LIN {X 0,Y 186.284,Z 510.696,A -85,B 0,C 180,E1 -23810.819,E2 -23810.819} C_VEL
LIN {X 0,Y 183.87,Z 513.938,A -85,B 0,C 180,E1 -23812.309,E2 -23812.309} C_VEL
LIN {X 0,Y 178.035,Z 519.948,A -85,B 0,C 180,E1 -23815.094,E2 -23815.094} C_VEL
LIN {X 0,Y 171.013,Z 526.327,A -85,B 0,C 180,E1 -23819.1,E2 -23819.1} C_VEL
LIN {X 0,Y 166.228,Z 530.269,A -85,B 0,C 180,E1 -23822.61,E2 -23822.61} C_VEL
LIN {X 0,Y 161.84,Z 533.649,A -85,B 0,C 180,E1 -23827.005,E2 -23827.005} C_VEL
LIN {X 0,Y 158.22,Z 535.815,A -85,B 0,C 180,E1 -23831.895,E2 -23831.895} C_VEL
LIN {X 0,Y 156.037,Z 536.613,A -85,B 0,C 180,E1 -23836.995,E2 -23836.995} C_VEL
LIN {X 0,Y 155.154,Z 536.037,A -85,B 0,C 180,E1 -23842.2,E2 -23842.2} C_VEL
LIN {X 0,Y 155.187,Z 535.075,A -85,B 0,C 180,E1 -23845.105,E2 -23845.105} C_VEL
LIN {X 0,Y 155.27,Z 533.944,A -85,B 0,C 180,E1 -23847.415,E2 -23847.415} C_VEL
LIN {X 0,Y 155.439,Z 531.27,A -85,B 0,C 180,E1 -23851.305,E2 -23851.305} C_VEL
LIN {X 0,Y 155.517,Z 527.484,A -85,B 0,C 180,E1 -23855.195,E2 -23855.195} C_VEL
LIN {X 0,Y 155.68,Z 522.461,A -85,B 0,C 180,E1 -23859.1,E2 -23859.1} C_VEL
LIN {X 0,Y 156.326,Z 516.101,A -85,B 0,C 180,E1 -23863,E2 -23863} C_VEL
LIN {X 0,Y 157.71,Z 508.216,A -85,B 0,C 180,E1 -23866.847,E2 -23866.847} C_VEL
LIN {X 0,Y 159.13,Z 500.124,A -85,B 0,C 180,E1 -23870.025,E2 -23870.025} C_VEL
LIN {X 0,Y 161.268,Z 490.423,A -85,B 0,C 180,E1 -23873.102,E2 -23873.102} C_VEL
LIN {X 0,Y 161.463,Z 485.361,A -85,B 0,C 180,E1 -23874.494,E2 -23874.494} C_VEL
LIN {X 0,Y 160.936,Z 473.75,A -85,B 0,C 180,E1 -23877.302,E2 -23877.302} C_VEL
LIN {X 0,Y 160.871,Z 471.959,A -85,B 0,C 180,E1 -23877.692,E2 -23877.692} C_VEL
LIN {X 0,Y 159.992,Z 466.935,A -85,B 0,C 180,E1 -23878.761,E2 -23878.761} C_VEL
LIN {X 0,Y 158.155,Z 462.064,A -85,B 0,C 180,E1 -23879.809,E2 -23879.809} C_VEL
LIN {X 0,Y 153.248,Z 450.597,A -85,B 0,C 180,E1 -23882.092,E2 -23882.092} C_VEL
LIN {X 0,Y 152.195,Z 445.196,A -85,B 0,C 180,E1 -23882.916,E2 -23882.916} C_VEL
LIN {X 0,Y 151.126,Z 432.472,A -85,B 0,C 180,E1 -23884.435,E2 -23884.435} C_VEL
LIN {X 0,Y 151.945,Z 429.73,A -85,B 0,C 180,E1 -23888.155,E2 -23888.155} C_VEL
LIN {X 0,Y 151.552,Z 426.949,A -85,B 0,C 180,E1 -23892.097,E2 -23892.097} C_VEL
LIN {X 0,Y 150.529,Z 422.213,A -85,B 0,C 180,E1 -23899.18,E2 -23899.18} C_VEL
LIN {X 0,Y 150.464,Z 421.742,A -85,B 0,C 180,E1 -23900.038,E2 -23900.038} C_VEL
LIN {X 0,Y 150.214,Z 421.77,A -85,B 0,C 180,E1 -23905.842,E2 -23905.842} C_VEL
LIN {X 0,Y 150.212,Z 421.775,A -85,B 0,C 180,E1 -23909.023,E2 -23909.023} C_VEL
LIN {X 0,Y 150.26,Z 421.764,A -85,B 0,C 180,E1 -23912.725,E2 -23912.725} C_VEL
LIN {X 0,Y 150.306,Z 421.761,A -85,B 0,C 180,E1 -23919.277,E2 -23919.277} C_VEL
LIN {X 0,Y 150.341,Z 421.756,A -85,B 0,C 180,E1 -23923.709,E2 -23923.709} C_VEL
LIN {X 0,Y 150.628,Z 421.717,A -85,B 0,C 180,E1 -23929.241,E2 -23929.241} C_VEL
LIN {X 0,Y 150.721,Z 421.708,A -85,B 0,C 180,E1 -23931.956,E2 -23931.956} C_VEL
LIN {X 0,Y 151.224,Z 421.644,A -85,B 0,C 180,E1 -23939.998,E2 -23939.998} C_VEL
LIN {X 0,Y 150.699,Z 421.709,A -85,B 0,C 180,E1 -23948.04,E2 -23948.04} C_VEL
LIN {X 0,Y 150.593,Z 421.726,A -85,B 0,C 180,E1 -23951.424,E2 -23951.424} C_VEL
LIN {X 0,Y 150.337,Z 421.754,A -85,B 0,C 180,E1 -23956.287,E2 -23956.287} C_VEL
LIN {X 0,Y 150.301,Z 421.763,A -85,B 0,C 180,E1 -23960.719,E2 -23960.719} C_VEL
LIN {X 0,Y 150.257,Z 421.768,A -85,B 0,C 180,E1 -23967.273,E2 -23967.273} C_VEL
LIN {X 0,Y 150.228,Z 421.767,A -85,B 0,C 180,E1 -23972.624,E2 -23972.624} C_VEL
LIN {X 0,Y 150.186,Z 421.775,A -85,B 0,C 180,E1 -23977.466,E2 -23977.466} C_VEL
LIN {X 0,Y 150.147,Z 421.778,A -85,B 0,C 180,E1 -23981.491,E2 -23981.491} C_VEL
LIN {X 0,Y 150.137,Z 421.782,A -85,B 0,C 180,E1 -23985.387,E2 -23985.387} C_VEL
LIN {X 0,Y 150.147,Z 421.778,A -85,B 0,C 180,E1 -23989.046,E2 -23989.046} C_VEL
LIN {X 0,Y 150.184,Z 421.778,A -85,B 0,C 180,E1 -23992.701,E2 -23992.701} C_VEL
LIN {X 0,Y 150.221,Z 421.767,A -85,B 0,C 180,E1 -23997.36,E2 -23997.36} C_VEL
LIN {X 0,Y 150.249,Z 421.768,A -85,B 0,C 180,E1 -24002.709,E2 -24002.709} C_VEL
LIN {X 0,Y 150.354,Z 421.755,A -85,B 0,C 180,E1 -24009.198,E2 -24009.198} C_VEL
LIN {X 0,Y 150.362,Z 421.749,A -85,B 0,C 180,E1 -24013.704,E2 -24013.704} C_VEL
LIN {X 0,Y 150.61,Z 421.723,A -85,B 0,C 180,E1 -24019.233,E2 -24019.233} C_VEL
LIN {X 0,Y 150.702,Z 421.708,A -85,B 0,C 180,E1 -24021.948,E2 -24021.948} C_VEL
LIN {X 0,Y 151.211,Z 421.645,A -85,B 0,C 180,E1 -24029.99,E2 -24029.99} C_VEL
LIN {X 0,Y 150.753,Z 421.702,A -85,B 0,C 180,E1 -24038.029,E2 -24038.029} C_VEL
LIN {X 0,Y 150.624,Z 421.721,A -85,B 0,C 180,E1 -24041.536,E2 -24041.536} C_VEL
LIN {X 0,Y 150.366,Z 421.749,A -85,B 0,C 180,E1 -24046.275,E2 -24046.275} C_VEL
LIN {X 0,Y 150.295,Z 421.763,A -85,B 0,C 180,E1 -24050.743,E2 -24050.743} C_VEL
LIN {X 0,Y 149.941,Z 421.807,A -85,B 0,C 180,E1 -24057.062,E2 -24057.062} C_VEL
LIN {X 0,Y 149.878,Z 421.816,A -85,B 0,C 180,E1 -24058.142,E2 -24058.142} C_VEL
LIN {X 0,Y 154.136,Z 437.425,A -85,B 0,C 180,E1 -24060.849,E2 -24060.849} C_VEL
LIN {X 0,Y 156.236,Z 448.528,A -85,B 0,C 180,E1 -24063.041,E2 -24063.041} C_VEL
LIN {X 0,Y 157.778,Z 458.692,A -85,B 0,C 180,E1 -24065.372,E2 -24065.372} C_VEL
LIN {X 0,Y 155.452,Z 470.191,A -85,B 0,C 180,E1 -24068.235,E2 -24068.235} C_VEL
LIN {X 0,Y 153.319,Z 480.244,A -85,B 0,C 180,E1 -24071.36,E2 -24071.36} C_VEL
LIN {X 0,Y 151.39,Z 489.245,A -85,B 0,C 180,E1 -24074.828,E2 -24074.828} C_VEL
LIN {X 0,Y 149.771,Z 497.763,A -85,B 0,C 180,E1 -24078.936,E2 -24078.936} C_VEL
LIN {X 0,Y 148.575,Z 505.298,A -85,B 0,C 180,E1 -24083.509,E2 -24083.509} C_VEL
LIN {X 0,Y 148.055,Z 509.738,A -85,B 0,C 180,E1 -24086.918,E2 -24086.918} C_VEL
LIN {X 0,Y 147.628,Z 514.587,A -85,B 0,C 180,E1 -24091.575,E2 -24091.575} C_VEL
LIN {X 0,Y 147.769,Z 517.072,A -85,B 0,C 180,E1 -24094.659,E2 -24094.659} C_VEL
LIN {X 0,Y 148.266,Z 519.046,A -85,B 0,C 180,E1 -24097.718,E2 -24097.718} C_VEL
LIN {X 0,Y 149.132,Z 520.547,A -85,B 0,C 180,E1 -24100.741,E2 -24100.741} C_VEL
LIN {X 0,Y 150.327,Z 521.525,A -85,B 0,C 180,E1 -24103.712,E2 -24103.712} C_VEL
LIN {X 0,Y 151.816,Z 522.077,A -85,B 0,C 180,E1 -24106.619,E2 -24106.619} C_VEL
LIN {X 0,Y 153.712,Z 522.204,A -85,B 0,C 180,E1 -24109.464,E2 -24109.464} C_VEL
LIN {X 0,Y 155.983,Z 521.83,A -85,B 0,C 180,E1 -24112.325,E2 -24112.325} C_VEL
LIN {X 0,Y 161.306,Z 519.905,A -85,B 0,C 180,E1 -24117.505,E2 -24117.505} C_VEL
LIN {X 0,Y 166.234,Z 517.262,A -85,B 0,C 180,E1 -24121.213,E2 -24121.213} C_VEL
LIN {X 0,Y 171.913,Z 513.503,A -85,B 0,C 180,E1 -24124.692,E2 -24124.692} C_VEL
LIN {X 0,Y 178.769,Z 508.097,A -85,B 0,C 180,E1 -24128.199,E2 -24128.199} C_VEL
LIN {X 0,Y 186.405,Z 501.052,A -85,B 0,C 180,E1 -24131.448,E2 -24131.448} C_VEL
LIN {X 0,Y 188.196,Z 499.207,A -85,B 0,C 180,E1 -24132.143,E2 -24132.143} C_VEL
LIN {X 0,Y 189.038,Z 497.92,A -85,B 0,C 180,E1 -24132.891,E2 -24132.891} C_VEL
LIN {X 0,Y 190.054,Z 495.282,A -85,B 0,C 180,E1 -24135.004,E2 -24135.004} C_VEL
LIN {X 0,Y 190.434,Z 493.141,A -85,B 0,C 180,E1 -24137.174,E2 -24137.174} C_VEL
LIN {X 0,Y 190.55,Z 491.468,A -85,B 0,C 180,E1 -24139.389,E2 -24139.389} C_VEL
LIN {X 0,Y 190.372,Z 489.734,A -85,B 0,C 180,E1 -24142.666,E2 -24142.666} C_VEL
LIN {X 0,Y 190.072,Z 488.922,A -85,B 0,C 180,E1 -24146.342,E2 -24146.342} C_VEL
LIN {X 0,Y 189.815,Z 489.084,A -85,B 0,C 180,E1 -24148.774,E2 -24148.774} C_VEL
LIN {X 0,Y 189.665,Z 490.589,A -85,B 0,C 180,E1 -24153.769,E2 -24153.769} C_VEL
LIN {X 0,Y 189.657,Z 492.192,A -85,B 0,C 180,E1 -24156.365,E2 -24156.365} C_VEL
LIN {X 0,Y 189.434,Z 494.597,A -85,B 0,C 180,E1 -24159.104,E2 -24159.104} C_VEL
LIN {X 0,Y 188.981,Z 497.907,A -85,B 0,C 180,E1 -24162.023,E2 -24162.023} C_VEL
LIN {X 0,Y 188.46,Z 499.443,A -85,B 0,C 180,E1 -24163.009,E2 -24163.009} C_VEL
LIN {X 0,Y 185.287,Z 505.48,A -85,B 0,C 180,E1 -24166.113,E2 -24166.113} C_VEL
LIN {X 0,Y 181.669,Z 511.043,A -85,B 0,C 180,E1 -24168.891,E2 -24168.891} C_VEL
LIN {X 0,Y 178.382,Z 515.174,A -85,B 0,C 180,E1 -24170.934,E2 -24170.934} C_VEL
LIN {X 0,Y 172.304,Z 520.809,A -85,B 0,C 180,E1 -24173.753,E2 -24173.753} C_VEL
LIN {X 0,Y 166.712,Z 525.49,A -85,B 0,C 180,E1 -24176.779,E2 -24176.779} C_VEL
LIN {X 0,Y 160.278,Z 530.311,A -85,B 0,C 180,E1 -24181.173,E2 -24181.173} C_VEL
LIN {X 0,Y 155.314,Z 533.608,A -85,B 0,C 180,E1 -24185.979,E2 -24185.979} C_VEL
LIN {X 0,Y 151.483,Z 535.547,A -85,B 0,C 180,E1 -24191.06,E2 -24191.06} C_VEL
LIN {X 0,Y 149.086,Z 536.131,A -85,B 0,C 180,E1 -24196.378,E2 -24196.378} C_VEL
LIN {X 0,Y 148.125,Z 535.287,A -85,B 0,C 180,E1 -24201.827,E2 -24201.827} C_VEL
LIN {X 0,Y 148.147,Z 534.138,A -85,B 0,C 180,E1 -24205.044,E2 -24205.044} C_VEL
LIN {X 0,Y 148.44,Z 531.257,A -85,B 0,C 180,E1 -24210.01,E2 -24210.01} C_VEL
LIN {X 0,Y 148.461,Z 527.636,A -85,B 0,C 180,E1 -24214.082,E2 -24214.082} C_VEL
LIN {X 0,Y 148.578,Z 522.822,A -85,B 0,C 180,E1 -24218.168,E2 -24218.168} C_VEL
LIN {X 0,Y 149.128,Z 516.697,A -85,B 0,C 180,E1 -24222.254,E2 -24222.254} C_VEL
LIN {X 0,Y 150.365,Z 509.043,A -85,B 0,C 180,E1 -24226.296,E2 -24226.296} C_VEL
LIN {X 0,Y 152.092,Z 499.536,A -85,B 0,C 180,E1 -24230.287,E2 -24230.287} C_VEL
LIN {X 0,Y 154.292,Z 489.859,A -85,B 0,C 180,E1 -24233.498,E2 -24233.498} C_VEL
LIN {X 0,Y 154.283,Z 482.243,A -85,B 0,C 180,E1 -24235.654,E2 -24235.654} C_VEL
LIN {X 0,Y 153.827,Z 471.757,A -85,B 0,C 180,E1 -24238.205,E2 -24238.205} C_VEL
LIN {X 0,Y 153.198,Z 459.294,A -85,B 0,C 180,E1 -24240.684,E2 -24240.684} C_VEL
LIN {X 0,Y 152.348,Z 447.028,A -85,B 0,C 180,E1 -24242.658,E2 -24242.658} C_VEL
LIN {X 0,Y 152.195,Z 445.196,A -85,B 0,C 180,E1 -24242.916,E2 -24242.916} C_VEL
LIN {X 0,Y 151.642,Z 441.74,A -85,B 0,C 180,E1 -24243.522,E2 -24243.522} C_VEL
LIN {X 0,Y 150.105,Z 437.288,A -85,B 0,C 180,E1 -24244.815,E2 -24244.815} C_VEL
LIN {X 0,Y 148.205,Z 433.717,A -85,B 0,C 180,E1 -24246.446,E2 -24246.446} C_VEL
LIN {X 0,Y 145.77,Z 430.041,A -85,B 0,C 180,E1 -24249.085,E2 -24249.085} C_VEL
LIN {X 0,Y 144.599,Z 428.036,A -85,B 0,C 180,E1 -24251.293,E2 -24251.293} C_VEL
LIN {X 0,Y 144.416,Z 427.493,A -85,B 0,C 180,E1 -24252.061,E2 -24252.061} C_VEL
LIN {X 0,Y 143.529,Z 423.298,A -85,B 0,C 180,E1 -24258.618,E2 -24258.618} C_VEL
LIN {X 0,Y 143.429,Z 422.618,A -85,B 0,C 180,E1 -24259.972,E2 -24259.972} C_VEL
LIN {X 0,Y 143.199,Z 422.647,A -85,B 0,C 180,E1 -24267.323,E2 -24267.323} C_VEL
LIN {X 0,Y 143.204,Z 422.643,A -85,B 0,C 180,E1 -24272.071,E2 -24272.071} C_VEL
LIN {X 0,Y 143.244,Z 422.642,A -85,B 0,C 180,E1 -24278.804,E2 -24278.804} C_VEL
LIN {X 0,Y 143.279,Z 422.633,A -85,B 0,C 180,E1 -24282.882,E2 -24282.882} C_VEL
LIN {X 0,Y 143.555,Z 422.6,A -85,B 0,C 180,E1 -24288.704,E2 -24288.704} C_VEL
LIN {X 0,Y 143.642,Z 422.59,A -85,B 0,C 180,E1 -24291.557,E2 -24291.557} C_VEL
LIN {X 0,Y 144.181,Z 422.522,A -85,B 0,C 180,E1 -24299.998,E2 -24299.998} C_VEL
LIN {X 0,Y 143.625,Z 422.591,A -85,B 0,C 180,E1 -24308.439,E2 -24308.439} C_VEL
LIN {X 0,Y 143.518,Z 422.607,A -85,B 0,C 180,E1 -24311.612,E2 -24311.612} C_VEL
LIN {X 0,Y 143.275,Z 422.637,A -85,B 0,C 180,E1 -24317.114,E2 -24317.114} C_VEL
LIN {X 0,Y 143.243,Z 422.64,A -85,B 0,C 180,E1 -24321.195,E2 -24321.195} C_VEL
LIN {X 0,Y 143.204,Z 422.646,A -85,B 0,C 180,E1 -24327.928,E2 -24327.928} C_VEL
LIN {X 0,Y 143.157,Z 422.65,A -85,B 0,C 180,E1 -24333.412,E2 -24333.412} C_VEL
LIN {X 0,Y 143.067,Z 422.658,A -85,B 0,C 180,E1 -24339.685,E2 -24339.685} C_VEL
LIN {X 0,Y 143.045,Z 422.665,A -85,B 0,C 180,E1 -24343.455,E2 -24343.455} C_VEL
LIN {X 0,Y 143.048,Z 422.662,A -85,B 0,C 180,E1 -24347.469,E2 -24347.469} C_VEL
LIN {X 0,Y 143.08,Z 422.661,A -85,B 0,C 180,E1 -24351.8,E2 -24351.8} C_VEL
LIN {X 0,Y 143.188,Z 422.643,A -85,B 0,C 180,E1 -24357.312,E2 -24357.312} C_VEL
LIN {X 0,Y 143.196,Z 422.648,A -85,B 0,C 180,E1 -24362.053,E2 -24362.053} C_VEL
LIN {X 0,Y 143.28,Z 422.637,A -85,B 0,C 180,E1 -24368.736,E2 -24368.736} C_VEL
LIN {X 0,Y 143.302,Z 422.629,A -85,B 0,C 180,E1 -24372.877,E2 -24372.877} C_VEL
LIN {X 0,Y 143.536,Z 422.605,A -85,B 0,C 180,E1 -24378.695,E2 -24378.695} C_VEL
LIN {X 0,Y 143.624,Z 422.59,A -85,B 0,C 180,E1 -24381.548,E2 -24381.548} C_VEL
LIN {X 0,Y 144.17,Z 422.522,A -85,B 0,C 180,E1 -24389.99,E2 -24389.99} C_VEL
LIN {X 0,Y 143.675,Z 422.583,A -85,B 0,C 180,E1 -24398.428,E2 -24398.428} C_VEL
LIN {X 0,Y 143.56,Z 422.602,A -85,B 0,C 180,E1 -24401.748,E2 -24401.748} C_VEL
LIN {X 0,Y 143.299,Z 422.628,A -85,B 0,C 180,E1 -24407.102,E2 -24407.102} C_VEL
LIN {X 0,Y 143.196,Z 422.647,A -85,B 0,C 180,E1 -24411.178,E2 -24411.178} C_VEL
LIN {X 0,Y 142.881,Z 422.687,A -85,B 0,C 180,E1 -24417.34,E2 -24417.34} C_VEL
LIN {X 0,Y 146.638,Z 436.414,A -85,B 0,C 180,E1 -24419.805,E2 -24419.805} C_VEL
LIN {X 0,Y 148.601,Z 445.45,A -85,B 0,C 180,E1 -24421.652,E2 -24421.652} C_VEL
LIN {X 0,Y 150.573,Z 457.441,A -85,B 0,C 180,E1 -24424.454,E2 -24424.454} C_VEL
LIN {X 0,Y 150.771,Z 458.859,A -85,B 0,C 180,E1 -24424.808,E2 -24424.808} C_VEL
LIN {X 0,Y 148.279,Z 471.16,A -85,B 0,C 180,E1 -24428.022,E2 -24428.022} C_VEL
LIN {X 0,Y 146.029,Z 481.475,A -85,B 0,C 180,E1 -24431.422,E2 -24431.422} C_VEL
LIN {X 0,Y 144.146,Z 490.189,A -85,B 0,C 180,E1 -24435.015,E2 -24435.015} C_VEL
LIN {X 0,Y 142.518,Z 498.703,A -85,B 0,C 180,E1 -24439.406,E2 -24439.406} C_VEL
LIN {X 0,Y 141.369,Z 506.139,A -85,B 0,C 180,E1 -24444.261,E2 -24444.261} C_VEL
LIN {X 0,Y 140.696,Z 511.785,A -85,B 0,C 180,E1 -24449.026,E2 -24449.026} C_VEL
LIN {X 0,Y 140.626,Z 516.35,A -85,B 0,C 180,E1 -24454.075,E2 -24454.075} C_VEL
LIN {X 0,Y 141.638,Z 519.928,A -85,B 0,C 180,E1 -24459.678,E2 -24459.678} C_VEL
LIN {X 0,Y 142.731,Z 521.268,A -85,B 0,C 180,E1 -24462.819,E2 -24462.819} C_VEL
LIN {X 0,Y 144.511,Z 522.324,A -85,B 0,C 180,E1 -24466.519,E2 -24466.519} C_VEL
LIN {X 0,Y 148.166,Z 522.652,A -85,B 0,C 180,E1 -24471.822,E2 -24471.822} C_VEL
LIN {X 0,Y 150.665,Z 522.238,A -85,B 0,C 180,E1 -24474.649,E2 -24474.649} C_VEL
LIN {X 0,Y 154.65,Z 520.992,A -85,B 0,C 180,E1 -24478.338,E2 -24478.338} C_VEL
LIN {X 0,Y 160.299,Z 518.379,A -85,B 0,C 180,E1 -24482.515,E2 -24482.515} C_VEL
LIN {X 0,Y 166.273,Z 514.894,A -85,B 0,C 180,E1 -24486.068,E2 -24486.068} C_VEL
LIN {X 0,Y 172.88,Z 510.246,A -85,B 0,C 180,E1 -24489.36,E2 -24489.36} C_VEL
LIN {X 0,Y 180.582,Z 503.877,A -85,B 0,C 180,E1 -24492.576,E2 -24492.576} C_VEL
LIN {X 0,Y 182.636,Z 501.98,A -85,B 0,C 180,E1 -24493.351,E2 -24493.351} C_VEL
LIN {X 0,Y 183.777,Z 500.455,A -85,B 0,C 180,E1 -24494.395,E2 -24494.395} C_VEL
LIN {X 0,Y 184.359,Z 499.237,A -85,B 0,C 180,E1 -24495.479,E2 -24495.479} C_VEL
LIN {X 0,Y 184.937,Z 496.956,A -85,B 0,C 180,E1 -24498.217,E2 -24498.217} C_VEL
LIN {X 0,Y 185.127,Z 495.825,A -85,B 0,C 180,E1 -24499.98,E2 -24499.98} C_VEL
LIN {X 0,Y 185.141,Z 494.707,A -85,B 0,C 180,E1 -24502.311,E2 -24502.311} C_VEL
LIN {X 0,Y 185.048,Z 494.058,A -85,B 0,C 180,E1 -24504.696,E2 -24504.696} C_VEL
LIN {X 0,Y 184.89,Z 493.877,A -85,B 0,C 180,E1 -24507.14,E2 -24507.14} C_VEL
LIN {X 0,Y 184.597,Z 494.24,A -85,B 0,C 180,E1 -24509.668,E2 -24509.668} C_VEL
LIN {X 0,Y 184.506,Z 495.274,A -85,B 0,C 180,E1 -24513.088,E2 -24513.088} C_VEL
LIN {X 0,Y 184.491,Z 496.09,A -85,B 0,C 180,E1 -24514.851,E2 -24514.851} C_VEL
LIN {X 0,Y 184.2,Z 498.085,A -85,B 0,C 180,E1 -24517.626,E2 -24517.626} C_VEL
LIN {X 0,Y 183.689,Z 500.93,A -85,B 0,C 180,E1 -24520.576,E2 -24520.576} C_VEL
LIN {X 0,Y 182.815,Z 503.139,A -85,B 0,C 180,E1 -24522.263,E2 -24522.263} C_VEL
LIN {X 0,Y 179.476,Z 508.433,A -85,B 0,C 180,E1 -24525.196,E2 -24525.196} C_VEL
LIN {X 0,Y 174.801,Z 514.4,A -85,B 0,C 180,E1 -24528.454,E2 -24528.454} C_VEL
LIN {X 0,Y 172.999,Z 516.318,A -85,B 0,C 180,E1 -24529.472,E2 -24529.472} C_VEL
LIN {X 0,Y 164.688,Z 523.261,A -85,B 0,C 180,E1 -24533.326,E2 -24533.326} C_VEL
LIN {X 0,Y 157.299,Z 528.475,A -85,B 0,C 180,E1 -24537.59,E2 -24537.59} C_VEL
LIN {X 0,Y 153.15,Z 531.143,A -85,B 0,C 180,E1 -24540.684,E2 -24540.684} C_VEL
LIN {X 0,Y 148.845,Z 533.576,A -85,B 0,C 180,E1 -24544.864,E2 -24544.864} C_VEL
LIN {X 0,Y 144.756,Z 535.251,A -85,B 0,C 180,E1 -24550.143,E2 -24550.143} C_VEL
LIN {X 0,Y 142.162,Z 535.549,A -85,B 0,C 180,E1 -24555.7,E2 -24555.7} C_VEL
LIN {X 0,Y 141.116,Z 534.515,A -85,B 0,C 180,E1 -24561.418,E2 -24561.418} C_VEL
LIN {X 0,Y 141.132,Z 533.221,A -85,B 0,C 180,E1 -24564.862,E2 -24564.862} C_VEL
LIN {X 0,Y 141.222,Z 532.023,A -85,B 0,C 180,E1 -24567.158,E2 -24567.158} C_VEL
LIN {X 0,Y 141.415,Z 528.997,A -85,B 0,C 180,E1 -24571.434,E2 -24571.434} C_VEL
LIN {X 0,Y 141.445,Z 524.811,A -85,B 0,C 180,E1 -24575.713,E2 -24575.713} C_VEL
LIN {X 0,Y 141.732,Z 519.36,A -85,B 0,C 180,E1 -24580.005,E2 -24580.005} C_VEL
LIN {X 0,Y 142.557,Z 512.448,A -85,B 0,C 180,E1 -24584.281,E2 -24584.281} C_VEL
LIN {X 0,Y 144.132,Z 503.901,A -85,B 0,C 180,E1 -24588.488,E2 -24588.488} C_VEL
LIN {X 0,Y 145.941,Z 495.208,A -85,B 0,C 180,E1 -24591.924,E2 -24591.924} C_VEL
LIN {X 0,Y 147.312,Z 489.121,A -85,B 0,C 180,E1 -24593.934,E2 -24593.934} C_VEL
LIN {X 0,Y 147.107,Z 478.462,A -85,B 0,C 180,E1 -24597.002,E2 -24597.002} C_VEL
LIN {X 0,Y 146.603,Z 466.518,A -85,B 0,C 180,E1 -24599.857,E2 -24599.857} C_VEL
LIN {X 0,Y 145.841,Z 453.798,A -85,B 0,C 180,E1 -24602.305,E2 -24602.305} C_VEL
LIN {X 0,Y 145.016,Z 441.745,A -85,B 0,C 180,E1 -24604.159,E2 -24604.159} C_VEL
LIN {X 0,Y 144.279,Z 432.046,A -85,B 0,C 180,E1 -24605.405,E2 -24605.405} C_VEL
LIN {X 0,Y 144.715,Z 430.692,A -85,B 0,C 180,E1 -24607.335,E2 -24607.335} C_VEL
LIN {X 0,Y 144.604,Z 428.185,A -85,B 0,C 180,E1 -24611.017,E2 -24611.017} C_VEL
LIN {X 0,Y 144.416,Z 427.493,A -85,B 0,C 180,E1 -24612.061,E2 -24612.061} C_VEL
LIN {X 0,Y 143.4,Z 426.13,A -85,B 0,C 180,E1 -24614.306,E2 -24614.306} C_VEL
LIN {X 0,Y 141.503,Z 425.054,A -85,B 0,C 180,E1 -24616.528,E2 -24616.528} C_VEL
LIN {X 0,Y 137.323,Z 423.764,A -85,B 0,C 180,E1 -24621.127,E2 -24621.127} C_VEL
LIN {X 0,Y 136.18,Z 423.536,A -85,B 0,C 180,E1 -24623.588,E2 -24623.588} C_VEL
LIN {X 0,Y 136.09,Z 423.522,A -85,B 0,C 180,E1 -24624.428,E2 -24624.428} C_VEL
LIN {X 0,Y 136.077,Z 423.535,A -85,B 0,C 180,E1 -24628.901,E2 -24628.901} C_VEL
LIN {X 0,Y 136.161,Z 423.52,A -85,B 0,C 180,E1 -24632.317,E2 -24632.317} C_VEL
LIN {X 0,Y 136.207,Z 423.519,A -85,B 0,C 180,E1 -24638.824,E2 -24638.824} C_VEL
LIN {X 0,Y 136.251,Z 423.514,A -85,B 0,C 180,E1 -24645.051,E2 -24645.051} C_VEL
LIN {X 0,Y 136.448,Z 423.486,A -85,B 0,C 180,E1 -24648.177,E2 -24648.177} C_VEL
LIN {X 0,Y 136.568,Z 423.469,A -85,B 0,C 180,E1 -24651.116,E2 -24651.116} C_VEL
LIN {X 0,Y 137.138,Z 423.399,A -85,B 0,C 180,E1 -24659.997,E2 -24659.997} C_VEL
LIN {X 0,Y 136.554,Z 423.473,A -85,B 0,C 180,E1 -24668.879,E2 -24668.879} C_VEL
LIN {X 0,Y 136.433,Z 423.489,A -85,B 0,C 180,E1 -24671.888,E2 -24671.888} C_VEL
LIN {X 0,Y 136.187,Z 423.519,A -85,B 0,C 180,E1 -24678.034,E2 -24678.034} C_VEL
LIN {X 0,Y 136.17,Z 423.52,A -85,B 0,C 180,E1 -24681.693,E2 -24681.693} C_VEL
LIN {X 0,Y 136.114,Z 423.531,A -85,B 0,C 180,E1 -24688.607,E2 -24688.607} C_VEL
LIN {X 0,Y 136.057,Z 423.537,A -85,B 0,C 180,E1 -24694.622,E2 -24694.622} C_VEL
LIN {X 0,Y 136.04,Z 423.534,A -85,B 0,C 180,E1 -24699.187,E2 -24699.187} C_VEL
LIN {X 0,Y 135.99,Z 423.544,A -85,B 0,C 180,E1 -24703.64,E2 -24703.64} C_VEL
LIN {X 0,Y 135.992,Z 423.541,A -85,B 0,C 180,E1 -24707.778,E2 -24707.778} C_VEL
LIN {X 0,Y 136.029,Z 423.539,A -85,B 0,C 180,E1 -24711.673,E2 -24711.673} C_VEL
LIN {X 0,Y 136.062,Z 423.533,A -85,B 0,C 180,E1 -24715.73,E2 -24715.73} C_VEL
LIN {X 0,Y 136.152,Z 423.525,A -85,B 0,C 180,E1 -24722.306,E2 -24722.306} C_VEL
LIN {X 0,Y 136.247,Z 423.513,A -85,B 0,C 180,E1 -24728.823,E2 -24728.823} C_VEL
LIN {X 0,Y 136.268,Z 423.508,A -85,B 0,C 180,E1 -24735.045,E2 -24735.045} C_VEL
LIN {X 0,Y 136.444,Z 423.49,A -85,B 0,C 180,E1 -24738.127,E2 -24738.127} C_VEL
LIN {X 0,Y 136.549,Z 423.47,A -85,B 0,C 180,E1 -24741.107,E2 -24741.107} C_VEL
LIN {X 0,Y 137.127,Z 423.399,A -85,B 0,C 180,E1 -24749.989,E2 -24749.989} C_VEL
LIN {X 0,Y 136.598,Z 423.464,A -85,B 0,C 180,E1 -24758.868,E2 -24758.868} C_VEL
LIN {X 0,Y 136.481,Z 423.484,A -85,B 0,C 180,E1 -24761.947,E2 -24761.947} C_VEL
LIN {X 0,Y 136.227,Z 423.511,A -85,B 0,C 180,E1 -24768.02,E2 -24768.02} C_VEL
LIN {X 0,Y 136.115,Z 423.53,A -85,B 0,C 180,E1 -24771.669,E2 -24771.669} C_VEL
LIN {X 0,Y 135.881,Z 423.559,A -85,B 0,C 180,E1 -24776.481,E2 -24776.481} C_VEL
LIN {X 0,Y 139.781,Z 437.742,A -85,B 0,C 180,E1 -24779.21,E2 -24779.21} C_VEL
LIN {X 0,Y 141.852,Z 447.503,A -85,B 0,C 180,E1 -24781.334,E2 -24781.334} C_VEL
LIN {X 0,Y 143.744,Z 459.465,A -85,B 0,C 180,E1 -24784.307,E2 -24784.307} C_VEL
LIN {X 0,Y 141.429,Z 470.576,A -85,B 0,C 180,E1 -24787.341,E2 -24787.341} C_VEL
LIN {X 0,Y 138.947,Z 481.521,A -85,B 0,C 180,E1 -24791.097,E2 -24791.097} C_VEL
LIN {X 0,Y 136.863,Z 491.106,A -85,B 0,C 180,E1 -24795.284,E2 -24795.284} C_VEL
LIN {X 0,Y 135.346,Z 498.916,A -85,B 0,C 180,E1 -24799.532,E2 -24799.532} C_VEL
LIN {X 0,Y 134.337,Z 505.511,A -85,B 0,C 180,E1 -24803.971,E2 -24803.971} C_VEL
LIN {X 0,Y 133.697,Z 510.675,A -85,B 0,C 180,E1 -24808.29,E2 -24808.29} C_VEL
LIN {X 0,Y 133.505,Z 515.502,A -85,B 0,C 180,E1 -24813.469,E2 -24813.469} C_VEL
LIN {X 0,Y 134.182,Z 519.004,A -85,B 0,C 180,E1 -24818.495,E2 -24818.495} C_VEL
LIN {X 0,Y 135.173,Z 520.723,A -85,B 0,C 180,E1 -24821.826,E2 -24821.826} C_VEL
LIN {X 0,Y 137.273,Z 522.416,A -85,B 0,C 180,E1 -24826.539,E2 -24826.539} C_VEL
LIN {X 0,Y 141.618,Z 523.212,A -85,B 0,C 180,E1 -24832.891,E2 -24832.891} C_VEL
LIN {X 0,Y 147.587,Z 522.142,A -85,B 0,C 180,E1 -24838.861,E2 -24838.861} C_VEL
LIN {X 0,Y 152.519,Z 520.375,A -85,B 0,C 180,E1 -24842.643,E2 -24842.643} C_VEL
LIN {X 0,Y 158.553,Z 517.489,A -85,B 0,C 180,E1 -24846.365,E2 -24846.365} C_VEL
LIN {X 0,Y 165.307,Z 513.467,A -85,B 0,C 180,E1 -24849.793,E2 -24849.793} C_VEL
LIN {X 0,Y 173.184,Z 507.89,A -85,B 0,C 180,E1 -24853.153,E2 -24853.153} C_VEL
LIN {X 0,Y 177.651,Z 504.216,A -85,B 0,C 180,E1 -24854.903,E2 -24854.903} C_VEL
LIN {X 0,Y 178.531,Z 502.959,A -85,B 0,C 180,E1 -24855.997,E2 -24855.997} C_VEL
LIN {X 0,Y 179.246,Z 501.254,A -85,B 0,C 180,E1 -24858.283,E2 -24858.283} C_VEL
LIN {X 0,Y 179.544,Z 499.95,A -85,B 0,C 180,E1 -24860.63,E2 -24860.63} C_VEL
LIN {X 0,Y 179.672,Z 499.068,A -85,B 0,C 180,E1 -24863.028,E2 -24863.028} C_VEL
LIN {X 0,Y 179.542,Z 498.591,A -85,B 0,C 180,E1 -24865.824,E2 -24865.824} C_VEL
LIN {X 0,Y 179.437,Z 498.647,A -85,B 0,C 180,E1 -24868.037,E2 -24868.037} C_VEL
LIN {X 0,Y 179.104,Z 500.037,A -85,B 0,C 180,E1 -24873.325,E2 -24873.325} C_VEL
LIN {X 0,Y 178.87,Z 501.566,A -85,B 0,C 180,E1 -24876.114,E2 -24876.114} C_VEL
LIN {X 0,Y 178.266,Z 503.943,A -85,B 0,C 180,E1 -24879.111,E2 -24879.111} C_VEL
LIN {X 0,Y 177.361,Z 506.191,A -85,B 0,C 180,E1 -24881.174,E2 -24881.174} C_VEL
LIN {X 0,Y 173.69,Z 511.07,A -85,B 0,C 180,E1 -24884.145,E2 -24884.145} C_VEL
LIN {X 0,Y 169.588,Z 515.679,A -85,B 0,C 180,E1 -24886.873,E2 -24886.873} C_VEL
LIN {X 0,Y 167.733,Z 517.489,A -85,B 0,C 180,E1 -24887.916,E2 -24887.916} C_VEL
LIN {X 0,Y 159.078,Z 523.951,A -85,B 0,C 180,E1 -24891.806,E2 -24891.806} C_VEL
LIN {X 0,Y 151.372,Z 528.865,A -85,B 0,C 180,E1 -24896.155,E2 -24896.155} C_VEL
LIN {X 0,Y 145.069,Z 532.284,A -85,B 0,C 180,E1 -24901.036,E2 -24901.036} C_VEL
LIN {X 0,Y 140.063,Z 534.345,A -85,B 0,C 180,E1 -24906.345,E2 -24906.345} C_VEL
LIN {X 0,Y 136.42,Z 535.082,A -85,B 0,C 180,E1 -24912.007,E2 -24912.007} C_VEL
LIN {X 0,Y 134.525,Z 534.505,A -85,B 0,C 180,E1 -24917.95,E2 -24917.95} C_VEL
LIN {X 0,Y 134.073,Z 532.52,A -85,B 0,C 180,E1 -24923.993,E2 -24923.993} C_VEL
LIN {X 0,Y 134.269,Z 530.02,A -85,B 0,C 180,E1 -24928.511,E2 -24928.511} C_VEL
LIN {X 0,Y 134.403,Z 527.731,A -85,B 0,C 180,E1 -24931.509,E2 -24931.509} C_VEL
LIN {X 0,Y 134.454,Z 523.32,A -85,B 0,C 180,E1 -24936.012,E2 -24936.012} C_VEL
LIN {X 0,Y 134.894,Z 516.539,A -85,B 0,C 180,E1 -24941.277,E2 -24941.277} C_VEL
LIN {X 0,Y 135.972,Z 509.149,A -85,B 0,C 180,E1 -24945.756,E2 -24945.756} C_VEL
LIN {X 0,Y 137.37,Z 501.616,A -85,B 0,C 180,E1 -24949.434,E2 -24949.434} C_VEL
LIN {X 0,Y 139.66,Z 491.549,A -85,B 0,C 180,E1 -24953.357,E2 -24953.357} C_VEL
LIN {X 0,Y 140.24,Z 488.903,A -85,B 0,C 180,E1 -24954.248,E2 -24954.248} C_VEL
LIN {X 0,Y 140.089,Z 479.07,A -85,B 0,C 180,E1 -24957.255,E2 -24957.255} C_VEL
LIN {X 0,Y 139.653,Z 467.465,A -85,B 0,C 180,E1 -24960.226,E2 -24960.226} C_VEL
LIN {X 0,Y 138.952,Z 454.862,A -85,B 0,C 180,E1 -24962.844,E2 -24962.844} C_VEL
LIN {X 0,Y 138.049,Z 441.217,A -85,B 0,C 180,E1 -24965.068,E2 -24965.068} C_VEL
LIN {X 0,Y 137.376,Z 431.705,A -85,B 0,C 180,E1 -24966.291,E2 -24966.291} C_VEL
LIN {X 0,Y 137.65,Z 430.713,A -85,B 0,C 180,E1 -24967.796,E2 -24967.796} C_VEL
LIN {X 0,Y 137.344,Z 428.081,A -85,B 0,C 180,E1 -24971.902,E2 -24971.902} C_VEL
LIN {X 0,Y 136.439,Z 423.699,A -85,B 0,C 180,E1 -24979.106,E2 -24979.106} C_VEL
LIN {X 0,Y 136.09,Z 423.522,A -85,B 0,C 180,E1 -24984.428,E2 -24984.428} C_VEL
LIN {X 0,Y 135.452,Z 423.612,A -85,B 0,C 180,E1 -24986.897,E2 -24986.897} C_VEL
LIN {X 0,Y 133.939,Z 423.813,A -85,B 0,C 180,E1 -24989.335,E2 -24989.335} C_VEL
LIN {X 0,Y 129.469,Z 424.369,A -85,B 0,C 180,E1 -24996.051,E2 -24996.051} C_VEL
LIN {X 0,Y 129.088,Z 424.404,A -85,B 0,C 180,E1 -24997.825,E2 -24997.825} C_VEL
LIN {X 0,Y 129.172,Z 424.393,A -85,B 0,C 180,E1 -25004.211,E2 -25004.211} C_VEL
LIN {X 0,Y 129.366,Z 424.368,A -85,B 0,C 180,E1 -25007.971,E2 -25007.971} C_VEL
LIN {X 0,Y 129.492,Z 424.348,A -85,B 0,C 180,E1 -25010.627,E2 -25010.627} C_VEL
LIN {X 0,Y 130.092,Z 424.276,A -85,B 0,C 180,E1 -25019.997,E2 -25019.997} C_VEL
LIN {X 0,Y 129.48,Z 424.356,A -85,B 0,C 180,E1 -25029.369,E2 -25029.369} C_VEL
LIN {X 0,Y 129.318,Z 424.376,A -85,B 0,C 180,E1 -25032.553,E2 -25032.553} C_VEL
LIN {X 0,Y 129.104,Z 424.403,A -85,B 0,C 180,E1 -25039.061,E2 -25039.061} C_VEL
LIN {X 0,Y 129.091,Z 424.401,A -85,B 0,C 180,E1 -25042.398,E2 -25042.398} C_VEL
LIN {X 0,Y 129.031,Z 424.41,A -85,B 0,C 180,E1 -25045.829,E2 -25045.829} C_VEL
LIN {X 0,Y 129.033,Z 424.41,A -85,B 0,C 180,E1 -25049.35,E2 -25049.35} C_VEL
LIN {X 0,Y 128.973,Z 424.419,A -85,B 0,C 180,E1 -25055.159,E2 -25055.159} C_VEL
LIN {X 0,Y 128.936,Z 424.419,A -85,B 0,C 180,E1 -25060.847,E2 -25060.847} C_VEL
LIN {X 0,Y 128.923,Z 424.425,A -85,B 0,C 180,E1 -25065.123,E2 -25065.123} C_VEL
LIN {X 0,Y 128.943,Z 424.418,A -85,B 0,C 180,E1 -25069.73,E2 -25069.73} C_VEL
LIN {X 0,Y 128.965,Z 424.418,A -85,B 0,C 180,E1 -25074.823,E2 -25074.823} C_VEL
LIN {X 0,Y 129.022,Z 424.414,A -85,B 0,C 180,E1 -25080.632,E2 -25080.632} C_VEL
LIN {X 0,Y 129.035,Z 424.408,A -85,B 0,C 180,E1 -25084.157,E2 -25084.157} C_VEL
LIN {X 0,Y 129.111,Z 424.4,A -85,B 0,C 180,E1 -25087.717,E2 -25087.717} C_VEL
LIN {X 0,Y 129.155,Z 424.395,A -85,B 0,C 180,E1 -25090.933,E2 -25090.933} C_VEL
LIN {X 0,Y 129.365,Z 424.371,A -85,B 0,C 180,E1 -25097.912,E2 -25097.912} C_VEL
LIN {X 0,Y 129.475,Z 424.353,A -85,B 0,C 180,E1 -25100.617,E2 -25100.617} C_VEL
LIN {X 0,Y 130.082,Z 424.276,A -85,B 0,C 180,E1 -25109.989,E2 -25109.989} C_VEL
LIN {X 0,Y 129.52,Z 424.345,A -85,B 0,C 180,E1 -25119.357,E2 -25119.357} C_VEL
LIN {X 0,Y 129.383,Z 424.368,A -85,B 0,C 180,E1 -25122.537,E2 -25122.537} C_VEL
LIN {X 0,Y 129.113,Z 424.399,A -85,B 0,C 180,E1 -25129.05,E2 -25129.05} C_VEL
LIN {X 0,Y 128.894,Z 424.427,A -85,B 0,C 180,E1 -25134.125,E2 -25134.125} C_VEL
LIN {X 0,Y 128.843,Z 424.435,A -85,B 0,C 180,E1 -25135.534,E2 -25135.534} C_VEL
LIN {X 0,Y 132.387,Z 436.919,A -85,B 0,C 180,E1 -25138.095,E2 -25138.095} C_VEL
LIN {X 0,Y 134.46,Z 446.131,A -85,B 0,C 180,E1 -25140.19,E2 -25140.19} C_VEL
LIN {X 0,Y 136.32,Z 457.304,A -85,B 0,C 180,E1 -25143.061,E2 -25143.061} C_VEL
LIN {X 0,Y 136.638,Z 459.484,A -85,B 0,C 180,E1 -25143.663,E2 -25143.663} C_VEL
LIN {X 0,Y 135.475,Z 465.785,A -85,B 0,C 180,E1 -25145.378,E2 -25145.378} C_VEL
LIN {X 0,Y 133.09,Z 476.479,A -85,B 0,C 180,E1 -25148.826,E2 -25148.826} C_VEL
LIN {X 0,Y 131.001,Z 485.361,A -85,B 0,C 180,E1 -25152.372,E2 -25152.372} C_VEL
LIN {X 0,Y 129.313,Z 493.093,A -85,B 0,C 180,E1 -25156.14,E2 -25156.14} C_VEL
LIN {X 0,Y 128.037,Z 499.944,A -85,B 0,C 180,E1 -25160.196,E2 -25160.196} C_VEL
LIN {X 0,Y 127.134,Z 505.915,A -85,B 0,C 180,E1 -25164.524,E2 -25164.524} C_VEL
LIN {X 0,Y 126.455,Z 511.955,A -85,B 0,C 180,E1 -25169.991,E2 -25169.991} C_VEL
LIN {X 0,Y 126.58,Z 516.522,A -85,B 0,C 180,E1 -25175.395,E2 -25175.395} C_VEL
LIN {X 0,Y 127.633,Z 519.88,A -85,B 0,C 180,E1 -25180.711,E2 -25180.711} C_VEL
LIN {X 0,Y 130.029,Z 522.362,A -85,B 0,C 180,E1 -25186.572,E2 -25186.572} C_VEL
LIN {X 0,Y 132.606,Z 523.412,A -85,B 0,C 180,E1 -25190.854,E2 -25190.854} C_VEL
LIN {X 0,Y 135.075,Z 523.697,A -85,B 0,C 180,E1 -25194.03,E2 -25194.03} C_VEL
LIN {X 0,Y 140.535,Z 523.166,A -85,B 0,C 180,E1 -25199.481,E2 -25199.481} C_VEL
LIN {X 0,Y 144.749,Z 522.053,A -85,B 0,C 180,E1 -25202.785,E2 -25202.785} C_VEL
LIN {X 0,Y 148.73,Z 520.627,A -85,B 0,C 180,E1 -25205.425,E2 -25205.425} C_VEL
LIN {X 0,Y 153.033,Z 518.776,A -85,B 0,C 180,E1 -25207.921,E2 -25207.921} C_VEL
LIN {X 0,Y 160.097,Z 515.069,A -85,B 0,C 180,E1 -25211.396,E2 -25211.396} C_VEL
LIN {X 0,Y 167.765,Z 510.149,A -85,B 0,C 180,E1 -25214.56,E2 -25214.56} C_VEL
LIN {X 0,Y 170.469,Z 508.208,A -85,B 0,C 180,E1 -25215.546,E2 -25215.546} C_VEL
LIN {X 0,Y 172.558,Z 506.499,A -85,B 0,C 180,E1 -25216.567,E2 -25216.567} C_VEL
LIN {X 0,Y 173.44,Z 504.983,A -85,B 0,C 180,E1 -25218.917,E2 -25218.917} C_VEL
LIN {X 0,Y 173.841,Z 503.791,A -85,B 0,C 180,E1 -25221.618,E2 -25221.618} C_VEL
LIN {X 0,Y 173.971,Z 503.24,A -85,B 0,C 180,E1 -25223.829,E2 -25223.829} C_VEL
LIN {X 0,Y 173.873,Z 503.017,A -85,B 0,C 180,E1 -25227.243,E2 -25227.243} C_VEL
LIN {X 0,Y 173.5,Z 503.935,A -85,B 0,C 180,E1 -25231.778,E2 -25231.778} C_VEL
LIN {X 0,Y 173.371,Z 504.975,A -85,B 0,C 180,E1 -25234.58,E2 -25234.58} C_VEL
LIN {X 0,Y 172.747,Z 506.97,A -85,B 0,C 180,E1 -25237.61,E2 -25237.61} C_VEL
LIN {X 0,Y 172.249,Z 508.223,A -85,B 0,C 180,E1 -25239.19,E2 -25239.19} C_VEL
LIN {X 0,Y 171.181,Z 509.897,A -85,B 0,C 180,E1 -25240.594,E2 -25240.594} C_VEL
LIN {X 0,Y 168.007,Z 513.454,A -85,B 0,C 180,E1 -25242.956,E2 -25242.956} C_VEL
LIN {X 0,Y 164.489,Z 516.911,A -85,B 0,C 180,E1 -25245.186,E2 -25245.186} C_VEL
LIN {X 0,Y 162.563,Z 518.566,A -85,B 0,C 180,E1 -25246.248,E2 -25246.248} C_VEL
LIN {X 0,Y 153.593,Z 524.663,A -85,B 0,C 180,E1 -25250.177,E2 -25250.177} C_VEL
LIN {X 0,Y 145.534,Z 529.174,A -85,B 0,C 180,E1 -25254.599,E2 -25254.599} C_VEL
LIN {X 0,Y 138.874,Z 532.291,A -85,B 0,C 180,E1 -25259.611,E2 -25259.611} C_VEL
LIN {X 0,Y 133.564,Z 534.096,A -85,B 0,C 180,E1 -25265.118,E2 -25265.118} C_VEL
LIN {X 0,Y 129.668,Z 534.558,A -85,B 0,C 180,E1 -25271.035,E2 -25271.035} C_VEL
LIN {X 0,Y 127.593,Z 533.712,A -85,B 0,C 180,E1 -25277.284,E2 -25277.284} C_VEL
LIN {X 0,Y 127.079,Z 531.5,A -85,B 0,C 180,E1 -25283.661,E2 -25283.661} C_VEL
LIN {X 0,Y 127.299,Z 528.814,A -85,B 0,C 180,E1 -25288.43,E2 -25288.43} C_VEL
LIN {X 0,Y 127.412,Z 526.442,A -85,B 0,C 180,E1 -25291.592,E2 -25291.592} C_VEL
LIN {X 0,Y 127.447,Z 521.795,A -85,B 0,C 180,E1 -25296.343,E2 -25296.343} C_VEL
LIN {X 0,Y 127.847,Z 515.833,A -85,B 0,C 180,E1 -25301.104,E2 -25301.104} C_VEL
LIN {X 0,Y 128.919,Z 508.358,A -85,B 0,C 180,E1 -25305.829,E2 -25305.829} C_VEL
LIN {X 0,Y 130.362,Z 500.767,A -85,B 0,C 180,E1 -25309.702,E2 -25309.702} C_VEL
LIN {X 0,Y 132.432,Z 491.663,A -85,B 0,C 180,E1 -25313.465,E2 -25313.465} C_VEL
LIN {X 0,Y 133.205,Z 487.395,A -85,B 0,C 180,E1 -25314.978,E2 -25314.978} C_VEL
LIN {X 0,Y 132.87,Z 476.383,A -85,B 0,C 180,E1 -25318.439,E2 -25318.439} C_VEL
LIN {X 0,Y 132.522,Z 464.824,A -85,B 0,C 180,E1 -25321.421,E2 -25321.421} C_VEL
LIN {X 0,Y 131.848,Z 451.124,A -85,B 0,C 180,E1 -25324.277,E2 -25324.277} C_VEL
LIN {X 0,Y 130.95,Z 437.607,A -85,B 0,C 180,E1 -25326.46,E2 -25326.46} C_VEL
LIN {X 0,Y 130.463,Z 431.329,A -85,B 0,C 180,E1 -25327.314,E2 -25327.314} C_VEL
LIN {X 0,Y 130.365,Z 429.076,A -85,B 0,C 180,E1 -25330.994,E2 -25330.994} C_VEL
LIN {X 0,Y 129.506,Z 425.406,A -85,B 0,C 180,E1 -25337.282,E2 -25337.282} C_VEL
LIN {X 0,Y 129.365,Z 424.371,A -85,B 0,C 180,E1 -25339.53,E2 -25339.53} C_VEL
LIN {X 0,Y 129.016,Z 424.411,A -85,B 0,C 180,E1 -25346.99,E2 -25346.99} C_VEL
LIN {X 0,Y 129.039,Z 424.411,A -85,B 0,C 180,E1 -25350.645,E2 -25350.645} C_VEL
LIN {X 0,Y 129.091,Z 424.404,A -85,B 0,C 180,E1 -25357.772,E2 -25357.772} C_VEL
LIN {X 0,Y 129.088,Z 424.404,A -85,B 0,C 180,E1 -25357.825,E2 -25357.825} C_VEL
LIN {X 0,Y 128.358,Z 424.493,A -85,B 0,C 180,E1 -25360.433,E2 -25360.433} C_VEL
LIN {X 0,Y 126.833,Z 424.683,A -85,B 0,C 180,E1 -25363.013,E2 -25363.013} C_VEL
LIN {X 0,Y 122.639,Z 425.201,A -85,B 0,C 180,E1 -25370.137,E2 -25370.137} C_VEL
LIN {X 0,Y 122.38,Z 425.231,A -85,B 0,C 180,E1 -25372.011,E2 -25372.011} C_VEL
LIN {X 0,Y 123.045,Z 425.154,A -85,B 0,C 180,E1 -25379.997,E2 -25379.997} C_VEL
LIN {X 0,Y 122.405,Z 425.23,A -85,B 0,C 180,E1 -25386.919,E2 -25386.919} C_VEL
LIN {X 0,Y 122.306,Z 425.25,A -85,B 0,C 180,E1 -25392.302,E2 -25392.302} C_VEL
LIN {X 0,Y 122.081,Z 425.274,A -85,B 0,C 180,E1 -25396.726,E2 -25396.726} C_VEL
LIN {X 0,Y 122.023,Z 425.279,A -85,B 0,C 180,E1 -25402.823,E2 -25402.823} C_VEL
LIN {X 0,Y 121.951,Z 425.294,A -85,B 0,C 180,E1 -25407.451,E2 -25407.451} C_VEL
LIN {X 0,Y 121.915,Z 425.292,A -85,B 0,C 180,E1 -25411.25,E2 -25411.25} C_VEL
LIN {X 0,Y 121.897,Z 425.301,A -85,B 0,C 180,E1 -25416.161,E2 -25416.161} C_VEL
LIN {X 0,Y 121.876,Z 425.3,A -85,B 0,C 180,E1 -25421.424,E2 -25421.424} C_VEL
LIN {X 0,Y 121.873,Z 425.298,A -85,B 0,C 180,E1 -25428.557,E2 -25428.557} C_VEL
LIN {X 0,Y 121.916,Z 425.296,A -85,B 0,C 180,E1 -25434.785,E2 -25434.785} C_VEL
LIN {X 0,Y 121.933,Z 425.295,A -85,B 0,C 180,E1 -25439.828,E2 -25439.828} C_VEL
LIN {X 0,Y 121.987,Z 425.284,A -85,B 0,C 180,E1 -25446.204,E2 -25446.204} C_VEL
LIN {X 0,Y 122.048,Z 425.282,A -85,B 0,C 180,E1 -25449.775,E2 -25449.775} C_VEL
LIN {X 0,Y 122.239,Z 425.258,A -85,B 0,C 180,E1 -25456.692,E2 -25456.692} C_VEL
LIN {X 0,Y 122.405,Z 425.235,A -85,B 0,C 180,E1 -25460.07,E2 -25460.07} C_VEL
LIN {X 0,Y 122.593,Z 425.214,A -85,B 0,C 180,E1 -25466.702,E2 -25466.702} C_VEL
LIN {X 0,Y 123.036,Z 425.153,A -85,B 0,C 180,E1 -25469.988,E2 -25469.988} C_VEL
LIN {X 0,Y 122.447,Z 425.23,A -85,B 0,C 180,E1 -25476.579,E2 -25476.579} C_VEL
LIN {X 0,Y 122.446,Z 425.228,A -85,B 0,C 180,E1 -25479.903,E2 -25479.903} C_VEL
LIN {X 0,Y 122.251,Z 425.256,A -85,B 0,C 180,E1 -25483.281,E2 -25483.281} C_VEL
LIN {X 0,Y 121.989,Z 425.29,A -85,B 0,C 180,E1 -25490.209,E2 -25490.209} C_VEL
LIN {X 0,Y 121.856,Z 425.436,A -85,B 0,C 180,E1 -25494.59,E2 -25494.59} C_VEL
LIN {X 0,Y 125.23,Z 437.116,A -85,B 0,C 180,E1 -25497.114,E2 -25497.114} C_VEL
LIN {X 0,Y 127.649,Z 447.74,A -85,B 0,C 180,E1 -25499.689,E2 -25499.689} C_VEL
LIN {X 0,Y 129.473,Z 459.207,A -85,B 0,C 180,E1 -25502.861,E2 -25502.861} C_VEL
LIN {X 0,Y 129.603,Z 460.806,A -85,B 0,C 180,E1 -25503.329,E2 -25503.329} C_VEL
LIN {X 0,Y 126.824,Z 473.397,A -85,B 0,C 180,E1 -25507.218,E2 -25507.218} C_VEL
LIN {X 0,Y 124.478,Z 482.928,A -85,B 0,C 180,E1 -25510.966,E2 -25510.966} C_VEL
LIN {X 0,Y 122.486,Z 491.811,A -85,B 0,C 180,E1 -25515.346,E2 -25515.346} C_VEL
LIN {X 0,Y 120.918,Z 499.837,A -85,B 0,C 180,E1 -25520.261,E2 -25520.261} C_VEL
LIN {X 0,Y 119.955,Z 506.193,A -85,B 0,C 180,E1 -25525.085,E2 -25525.085} C_VEL
LIN {X 0,Y 119.382,Z 511.402,A -85,B 0,C 180,E1 -25529.978,E2 -25529.978} C_VEL
LIN {X 0,Y 119.528,Z 516.2,A -85,B 0,C 180,E1 -25535.699,E2 -25535.699} C_VEL
LIN {X 0,Y 120.185,Z 518.708,A -85,B 0,C 180,E1 -25539.463,E2 -25539.463} C_VEL
LIN {X 0,Y 121.283,Z 520.693,A -85,B 0,C 180,E1 -25543.161,E2 -25543.161} C_VEL
LIN {X 0,Y 122.862,Z 522.249,A -85,B 0,C 180,E1 -25546.776,E2 -25546.776} C_VEL
LIN {X 0,Y 124.836,Z 523.35,A -85,B 0,C 180,E1 -25550.279,E2 -25550.279} C_VEL
LIN {X 0,Y 127.252,Z 523.987,A -85,B 0,C 180,E1 -25553.661,E2 -25553.661} C_VEL
LIN {X 0,Y 130.086,Z 524.222,A -85,B 0,C 180,E1 -25556.906,E2 -25556.906} C_VEL
LIN {X 0,Y 133.502,Z 524.036,A -85,B 0,C 180,E1 -25560.171,E2 -25560.171} C_VEL
LIN {X 0,Y 140.945,Z 522.386,A -85,B 0,C 180,E1 -25565.726,E2 -25565.726} C_VEL
LIN {X 0,Y 145.327,Z 520.927,A -85,B 0,C 180,E1 -25568.344,E2 -25568.344} C_VEL
LIN {X 0,Y 152.624,Z 517.779,A -85,B 0,C 180,E1 -25572.039,E2 -25572.039} C_VEL
LIN {X 0,Y 160.254,Z 513.668,A -85,B 0,C 180,E1 -25575.258,E2 -25575.258} C_VEL
LIN {X 0,Y 165.833,Z 510.163,A -85,B 0,C 180,E1 -25577.259,E2 -25577.259} C_VEL
LIN {X 0,Y 167.489,Z 508.485,A -85,B 0,C 180,E1 -25579.616,E2 -25579.616} C_VEL
LIN {X 0,Y 168.007,Z 507.41,A -85,B 0,C 180,E1 -25583.057,E2 -25583.057} C_VEL
LIN {X 0,Y 168.075,Z 507.137,A -85,B 0,C 180,E1 -25587.387,E2 -25587.387} C_VEL
LIN {X 0,Y 167.776,Z 507.609,A -85,B 0,C 180,E1 -25590.179,E2 -25590.179} C_VEL
LIN {X 0,Y 167.573,Z 508.476,A -85,B 0,C 180,E1 -25593.042,E2 -25593.042} C_VEL
LIN {X 0,Y 166.892,Z 510.424,A -85,B 0,C 180,E1 -25596.877,E2 -25596.877} C_VEL
LIN {X 0,Y 166.248,Z 511.667,A -85,B 0,C 180,E1 -25598.568,E2 -25598.568} C_VEL
LIN {X 0,Y 164.918,Z 513.222,A -85,B 0,C 180,E1 -25599.924,E2 -25599.924} C_VEL
LIN {X 0,Y 161.409,Z 516.506,A -85,B 0,C 180,E1 -25602.267,E2 -25602.267} C_VEL
LIN {X 0,Y 157.533,Z 519.629,A -85,B 0,C 180,E1 -25604.47,E2 -25604.47} C_VEL
LIN {X 0,Y 148.247,Z 525.279,A -85,B 0,C 180,E1 -25608.432,E2 -25608.432} C_VEL
LIN {X 0,Y 139.825,Z 529.474,A -85,B 0,C 180,E1 -25612.918,E2 -25612.918} C_VEL
LIN {X 0,Y 132.762,Z 532.271,A -85,B 0,C 180,E1 -25618.051,E2 -25618.051} C_VEL
LIN {X 0,Y 127.138,Z 533.757,A -85,B 0,C 180,E1 -25623.768,E2 -25623.768} C_VEL
LIN {X 0,Y 122.963,Z 533.956,A -85,B 0,C 180,E1 -25629.958,E2 -25629.958} C_VEL
LIN {X 0,Y 120.685,Z 532.882,A -85,B 0,C 180,E1 -25636.543,E2 -25636.543} C_VEL
LIN {X 0,Y 120.092,Z 530.448,A -85,B 0,C 180,E1 -25643.291,E2 -25643.291} C_VEL
LIN {X 0,Y 120.321,Z 527.574,A -85,B 0,C 180,E1 -25648.339,E2 -25648.339} C_VEL
LIN {X 0,Y 120.438,Z 525.03,A -85,B 0,C 180,E1 -25651.684,E2 -25651.684} C_VEL
LIN {X 0,Y 120.465,Z 520.159,A -85,B 0,C 180,E1 -25656.713,E2 -25656.713} C_VEL
LIN {X 0,Y 120.934,Z 513.934,A -85,B 0,C 180,E1 -25661.748,E2 -25661.748} C_VEL
LIN {X 0,Y 122.171,Z 506.162,A -85,B 0,C 180,E1 -25666.728,E2 -25666.728} C_VEL
LIN {X 0,Y 123.714,Z 498.221,A -85,B 0,C 180,E1 -25670.809,E2 -25670.809} C_VEL
LIN {X 0,Y 126.041,Z 488.738,A -85,B 0,C 180,E1 -25674.733,E2 -25674.733} C_VEL
LIN {X 0,Y 125.964,Z 479.661,A -85,B 0,C 180,E1 -25677.88,E2 -25677.88} C_VEL
LIN {X 0,Y 125.585,Z 467.441,A -85,B 0,C 180,E1 -25681.413,E2 -25681.413} C_VEL
LIN {X 0,Y 125.081,Z 454.737,A -85,B 0,C 180,E1 -25684.404,E2 -25684.404} C_VEL
LIN {X 0,Y 124.395,Z 441.702,A -85,B 0,C 180,E1 -25686.822,E2 -25686.822} C_VEL
LIN {X 0,Y 123.615,Z 432.513,A -85,B 0,C 180,E1 -25688.212,E2 -25688.212} C_VEL
LIN {X 0,Y 123.432,Z 430.925,A -85,B 0,C 180,E1 -25688.46,E2 -25688.46} C_VEL
LIN {X 0,Y 122.946,Z 428.173,A -85,B 0,C 180,E1 -25693.326,E2 -25693.326} C_VEL
LIN {X 0,Y 122.336,Z 425.247,A -85,B 0,C 180,E1 -25698.95,E2 -25698.95} C_VEL
LIN {X 0,Y 122.014,Z 425.28,A -85,B 0,C 180,E1 -25704.827,E2 -25704.827} C_VEL
LIN {X 0,Y 121.952,Z 425.293,A -85,B 0,C 180,E1 -25709.84,E2 -25709.84} C_VEL
LIN {X 0,Y 122.009,Z 425.288,A -85,B 0,C 180,E1 -25717.193,E2 -25717.193} C_VEL
LIN {X 0,Y 122.084,Z 425.274,A -85,B 0,C 180,E1 -25723.269,E2 -25723.269} C_VEL
LIN {X 0,Y 122.31,Z 425.247,A -85,B 0,C 180,E1 -25727.69,E2 -25727.69} C_VEL
LIN {X 0,Y 122.38,Z 425.231,A -85,B 0,C 180,E1 -25732.011,E2 -25732.011} C_VEL
LIN {X 0,Y 121.782,Z 425.317,A -85,B 0,C 180,E1 -25734.767,E2 -25734.767} C_VEL
LIN {X 0,Y 120.294,Z 425.51,A -85,B 0,C 180,E1 -25737.494,E2 -25737.494} C_VEL
LIN {X 0,Y 115.785,Z 426.066,A -85,B 0,C 180,E1 -25745.032,E2 -25745.032} C_VEL
LIN {X 0,Y 115.364,Z 426.108,A -85,B 0,C 180,E1 -25747.029,E2 -25747.029} C_VEL
LIN {X 0,Y 115.224,Z 426.132,A -85,B 0,C 180,E1 -25752.552,E2 -25752.552} C_VEL
LIN {X 0,Y 114.986,Z 426.16,A -85,B 0,C 180,E1 -25757.791,E2 -25757.791} C_VEL
LIN {X 0,Y 114.946,Z 426.159,A -85,B 0,C 180,E1 -25763.462,E2 -25763.462} C_VEL
LIN {X 0,Y 114.872,Z 426.17,A -85,B 0,C 180,E1 -25771.048,E2 -25771.048} C_VEL
LIN {X 0,Y 114.79,Z 426.185,A -85,B 0,C 180,E1 -25777.748,E2 -25777.748} C_VEL
LIN {X 0,Y 114.791,Z 426.185,A -85,B 0,C 180,E1 -25782.702,E2 -25782.702} C_VEL
LIN {X 0,Y 114.796,Z 426.181,A -85,B 0,C 180,E1 -25787.651,E2 -25787.651} C_VEL
LIN {X 0,Y 114.793,Z 426.186,A -85,B 0,C 180,E1 -25792.735,E2 -25792.735} C_VEL
LIN {X 0,Y 114.862,Z 426.176,A -85,B 0,C 180,E1 -25798.931,E2 -25798.931} C_VEL
LIN {X 0,Y 114.952,Z 426.161,A -85,B 0,C 180,E1 -25806.494,E2 -25806.494} C_VEL
LIN {X 0,Y 115.013,Z 426.154,A -85,B 0,C 180,E1 -25812.197,E2 -25812.197} C_VEL
LIN {X 0,Y 115.251,Z 426.128,A -85,B 0,C 180,E1 -25817.321,E2 -25817.321} C_VEL
LIN {X 0,Y 115.362,Z 426.111,A -85,B 0,C 180,E1 -25822.989,E2 -25822.989} C_VEL
LIN {X 0,Y 115.987,Z 426.031,A -85,B 0,C 180,E1 -25829.987,E2 -25829.987} C_VEL
LIN {X 0,Y 115.388,Z 426.108,A -85,B 0,C 180,E1 -25836.984,E2 -25836.984} C_VEL
LIN {X 0,Y 115.382,Z 426.11,A -85,B 0,C 180,E1 -25840.516,E2 -25840.516} C_VEL
LIN {X 0,Y 115.133,Z 426.143,A -85,B 0,C 180,E1 -25844.119,E2 -25844.119} C_VEL
LIN {X 0,Y 114.983,Z 426.155,A -85,B 0,C 180,E1 -25847.781,E2 -25847.781} C_VEL
LIN {X 0,Y 114.86,Z 426.333,A -85,B 0,C 180,E1 -25853.503,E2 -25853.503} C_VEL
LIN {X 0,Y 118.43,Z 438.658,A -85,B 0,C 180,E1 -25856.413,E2 -25856.413} C_VEL
LIN {X 0,Y 120.848,Z 449.569,A -85,B 0,C 180,E1 -25859.275,E2 -25859.275} C_VEL
LIN {X 0,Y 122.547,Z 460.515,A -85,B 0,C 180,E1 -25862.508,E2 -25862.508} C_VEL
LIN {X 0,Y 121.054,Z 467.871,A -85,B 0,C 180,E1 -25864.78,E2 -25864.78} C_VEL
LIN {X 0,Y 118.408,Z 478.803,A -85,B 0,C 180,E1 -25868.834,E2 -25868.834} C_VEL
LIN {X 0,Y 116.074,Z 488.471,A -85,B 0,C 180,E1 -25873.405,E2 -25873.405} C_VEL
LIN {X 0,Y 114.242,Z 497.231,A -85,B 0,C 180,E1 -25878.604,E2 -25878.604} C_VEL
LIN {X 0,Y 113.06,Z 504.362,A -85,B 0,C 180,E1 -25883.886,E2 -25883.886} C_VEL
LIN {X 0,Y 112.332,Z 510.789,A -85,B 0,C 180,E1 -25889.97,E2 -25889.97} C_VEL
LIN {X 0,Y 112.473,Z 515.787,A -85,B 0,C 180,E1 -25896.04,E2 -25896.04} C_VEL
LIN {X 0,Y 113.703,Z 519.581,A -85,B 0,C 180,E1 -25902.001,E2 -25902.001} C_VEL
LIN {X 0,Y 115.523,Z 521.869,A -85,B 0,C 180,E1 -25906.688,E2 -25906.688} C_VEL
LIN {X 0,Y 119.432,Z 523.968,A -85,B 0,C 180,E1 -25913.244,E2 -25913.244} C_VEL
LIN {X 0,Y 122.217,Z 524.56,A -85,B 0,C 180,E1 -25916.706,E2 -25916.706} C_VEL
LIN {X 0,Y 126.492,Z 524.716,A -85,B 0,C 180,E1 -25920.955,E2 -25920.955} C_VEL
LIN {X 0,Y 133.174,Z 523.833,A -85,B 0,C 180,E1 -25926.061,E2 -25926.061} C_VEL
LIN {X 0,Y 137.575,Z 522.75,A -85,B 0,C 180,E1 -25928.818,E2 -25928.818} C_VEL
LIN {X 0,Y 143.697,Z 520.714,A -85,B 0,C 180,E1 -25932.052,E2 -25932.052} C_VEL
LIN {X 0,Y 152.783,Z 516.774,A -85,B 0,C 180,E1 -25936.024,E2 -25936.024} C_VEL
LIN {X 0,Y 158.414,Z 513.803,A -85,B 0,C 180,E1 -25938.095,E2 -25938.095} C_VEL
LIN {X 0,Y 160.605,Z 512.43,A -85,B 0,C 180,E1 -25939.162,E2 -25939.162} C_VEL
LIN {X 0,Y 161.428,Z 511.767,A -85,B 0,C 180,E1 -25940.385,E2 -25940.385} C_VEL
LIN {X 0,Y 161.923,Z 511.089,A -85,B 0,C 180,E1 -25942.996,E2 -25942.996} C_VEL
LIN {X 0,Y 161.989,Z 510.889,A -85,B 0,C 180,E1 -25945.715,E2 -25945.715} C_VEL
LIN {X 0,Y 161.947,Z 511.07,A -85,B 0,C 180,E1 -25948.516,E2 -25948.516} C_VEL
LIN {X 0,Y 161.613,Z 511.756,A -85,B 0,C 180,E1 -25951.458,E2 -25951.458} C_VEL
LIN {X 0,Y 161.146,Z 512.87,A -85,B 0,C 180,E1 -25954.541,E2 -25954.541} C_VEL
LIN {X 0,Y 160.049,Z 514.885,A -85,B 0,C 180,E1 -25957.937,E2 -25957.937} C_VEL
LIN {X 0,Y 158.47,Z 516.274,A -85,B 0,C 180,E1 -25959.182,E2 -25959.182} C_VEL
LIN {X 0,Y 154.704,Z 519.197,A -85,B 0,C 180,E1 -25961.463,E2 -25961.463} C_VEL
LIN {X 0,Y 152.659,Z 520.643,A -85,B 0,C 180,E1 -25962.574,E2 -25962.574} C_VEL
LIN {X 0,Y 143.051,Z 525.874,A -85,B 0,C 180,E1 -25966.559,E2 -25966.559} C_VEL
LIN {X 0,Y 134.227,Z 529.69,A -85,B 0,C 180,E1 -25971.09,E2 -25971.09} C_VEL
LIN {X 0,Y 126.762,Z 532.173,A -85,B 0,C 180,E1 -25976.344,E2 -25976.344} C_VEL
LIN {X 0,Y 120.791,Z 533.397,A -85,B 0,C 180,E1 -25982.274,E2 -25982.274} C_VEL
LIN {X 0,Y 116.31,Z 533.325,A -85,B 0,C 180,E1 -25988.758,E2 -25988.758} C_VEL
LIN {X 0,Y 113.806,Z 531.965,A -85,B 0,C 180,E1 -25995.713,E2 -25995.713} C_VEL
LIN {X 0,Y 113.112,Z 529.274,A -85,B 0,C 180,E1 -26002.875,E2 -26002.875} C_VEL
LIN {X 0,Y 113.369,Z 526.239,A -85,B 0,C 180,E1 -26008.237,E2 -26008.237} C_VEL
LIN {X 0,Y 113.459,Z 523.55,A -85,B 0,C 180,E1 -26011.788,E2 -26011.788} C_VEL
LIN {X 0,Y 113.488,Z 518.41,A -85,B 0,C 180,E1 -26017.127,E2 -26017.127} C_VEL
LIN {X 0,Y 113.998,Z 511.882,A -85,B 0,C 180,E1 -26022.474,E2 -26022.474} C_VEL
LIN {X 0,Y 115.449,Z 503.782,A -85,B 0,C 180,E1 -26027.734,E2 -26027.734} C_VEL
LIN {X 0,Y 117.588,Z 493.672,A -85,B 0,C 180,E1 -26032.874,E2 -26032.874} C_VEL
LIN {X 0,Y 119.039,Z 487.698,A -85,B 0,C 180,E1 -26035.356,E2 -26035.356} C_VEL
LIN {X 0,Y 118.781,Z 476.872,A -85,B 0,C 180,E1 -26039.231,E2 -26039.231} C_VEL
LIN {X 0,Y 118.51,Z 464.967,A -85,B 0,C 180,E1 -26042.752,E2 -26042.752} C_VEL
LIN {X 0,Y 118.038,Z 451.407,A -85,B 0,C 180,E1 -26045.951,E2 -26045.951} C_VEL
LIN {X 0,Y 117.421,Z 439.259,A -85,B 0,C 180,E1 -26048.232,E2 -26048.232} C_VEL
LIN {X 0,Y 116.723,Z 433.049,A -85,B 0,C 180,E1 -26049.244,E2 -26049.244} C_VEL
LIN {X 0,Y 116.213,Z 430.531,A -85,B 0,C 180,E1 -26049.692,E2 -26049.692} C_VEL
LIN {X 0,Y 115.851,Z 428.631,A -85,B 0,C 180,E1 -26053.279,E2 -26053.279} C_VEL
LIN {X 0,Y 115.3,Z 426.124,A -85,B 0,C 180,E1 -26058.477,E2 -26058.477} C_VEL
LIN {X 0,Y 115.019,Z 426.157,A -85,B 0,C 180,E1 -26062.611,E2 -26062.611} C_VEL
LIN {X 0,Y 114.885,Z 426.175,A -85,B 0,C 180,E1 -26068.941,E2 -26068.941} C_VEL
LIN {X 0,Y 114.932,Z 426.168,A -85,B 0,C 180,E1 -26076.554,E2 -26076.554} C_VEL
LIN {X 0,Y 114.989,Z 426.155,A -85,B 0,C 180,E1 -26082.203,E2 -26082.203} C_VEL
LIN {X 0,Y 115.331,Z 426.112,A -85,B 0,C 180,E1 -26089.463,E2 -26089.463} C_VEL
LIN {X 0,Y 115.535,Z 426.091,A -85,B 0,C 180,E1 -26096.509,E2 -26096.509} C_VEL
LIN {X 0,Y 115.996,Z 426.032,A -85,B 0,C 180,E1 -26099.997,E2 -26099.997} C_VEL
LIN {X 0,Y 115.364,Z 426.108,A -85,B 0,C 180,E1 -26107.029,E2 -26107.029} C_VEL
LIN {X 0,Y 114.491,Z 426.224,A -85,B 0,C 180,E1 -26109.933,E2 -26109.933} C_VEL
LIN {X 0,Y 112.738,Z 426.44,A -85,B 0,C 180,E1 -26112.797,E2 -26112.797} C_VEL
LIN {X 0,Y 108.87,Z 426.924,A -85,B 0,C 180,E1 -26118.704,E2 -26118.704} C_VEL
LIN {X 0,Y 107.92,Z 427.039,A -85,B 0,C 180,E1 -26121.85,E2 -26121.85} C_VEL
LIN {X 0,Y 107.902,Z 427.037,A -85,B 0,C 180,E1 -26122.916,E2 -26122.916} C_VEL
LIN {X 0,Y 107.762,Z 427.062,A -85,B 0,C 180,E1 -26127.159,E2 -26127.159} C_VEL
LIN {X 0,Y 107.795,Z 427.05,A -85,B 0,C 180,E1 -26132.029,E2 -26132.029} C_VEL
LIN {X 0,Y 107.698,Z 427.066,A -85,B 0,C 180,E1 -26138.437,E2 -26138.437} C_VEL
LIN {X 0,Y 107.68,Z 427.071,A -85,B 0,C 180,E1 -26145.88,E2 -26145.88} C_VEL
LIN {X 0,Y 107.692,Z 427.069,A -85,B 0,C 180,E1 -26151.541,E2 -26151.541} C_VEL
LIN {X 0,Y 107.799,Z 427.053,A -85,B 0,C 180,E1 -26158.548,E2 -26158.548} C_VEL
LIN {X 0,Y 107.916,Z 427.04,A -85,B 0,C 180,E1 -26166.985,E2 -26166.985} C_VEL
LIN {X 0,Y 108.031,Z 427.024,A -85,B 0,C 180,E1 -26174.903,E2 -26174.903} C_VEL
LIN {X 0,Y 108.252,Z 427,A -85,B 0,C 180,E1 -26178.755,E2 -26178.755} C_VEL
LIN {X 0,Y 108.442,Z 426.978,A -85,B 0,C 180,E1 -26186.271,E2 -26186.271} C_VEL
LIN {X 0,Y 108.937,Z 426.909,A -85,B 0,C 180,E1 -26189.986,E2 -26189.986} C_VEL
LIN {X 0,Y 108.331,Z 426.987,A -85,B 0,C 180,E1 -26197.441,E2 -26197.441} C_VEL
LIN {X 0,Y 108.191,Z 427.008,A -85,B 0,C 180,E1 -26203.012,E2 -26203.012} C_VEL
LIN {X 0,Y 107.853,Z 427.05,A -85,B 0,C 180,E1 -26210.986,E2 -26210.986} C_VEL
LIN {X 0,Y 107.831,Z 427.052,A -85,B 0,C 180,E1 -26212.246,E2 -26212.246} C_VEL
LIN {X 0,Y 111.519,Z 439.655,A -85,B 0,C 180,E1 -26215.485,E2 -26215.485} C_VEL
LIN {X 0,Y 114.036,Z 451.199,A -85,B 0,C 180,E1 -26218.766,E2 -26218.766} C_VEL
LIN {X 0,Y 115.437,Z 460.682,A -85,B 0,C 180,E1 -26221.781,E2 -26221.781} C_VEL
LIN {X 0,Y 115.251,Z 463.105,A -85,B 0,C 180,E1 -26222.568,E2 -26222.568} C_VEL
LIN {X 0,Y 112.568,Z 474.076,A -85,B 0,C 180,E1 -26226.419,E2 -26226.419} C_VEL
LIN {X 0,Y 109.804,Z 484.796,A -85,B 0,C 180,E1 -26231.236,E2 -26231.236} C_VEL
LIN {X 0,Y 107.724,Z 493.931,A -85,B 0,C 180,E1 -26236.491,E2 -26236.491} C_VEL
LIN {X 0,Y 106.34,Z 501.432,A -85,B 0,C 180,E1 -26241.892,E2 -26241.892} C_VEL
LIN {X 0,Y 105.439,Z 508.005,A -85,B 0,C 180,E1 -26247.78,E2 -26247.78} C_VEL
LIN {X 0,Y 105.238,Z 513.724,A -85,B 0,C 180,E1 -26254.277,E2 -26254.277} C_VEL
LIN {X 0,Y 106.188,Z 518.126,A -85,B 0,C 180,E1 -26260.679,E2 -26260.679} C_VEL
LIN {X 0,Y 108.286,Z 521.324,A -85,B 0,C 180,E1 -26266.72,E2 -26266.72} C_VEL
LIN {X 0,Y 112.911,Z 524.179,A -85,B 0,C 180,E1 -26274.649,E2 -26274.649} C_VEL
LIN {X 0,Y 119.508,Z 525.247,A -85,B 0,C 180,E1 -26281.842,E2 -26281.842} C_VEL
LIN {X 0,Y 127.731,Z 524.651,A -85,B 0,C 180,E1 -26288.044,E2 -26288.044} C_VEL
LIN {X 0,Y 137.186,Z 522.399,A -85,B 0,C 180,E1 -26293.309,E2 -26293.309} C_VEL
LIN {X 0,Y 145.254,Z 519.526,A -85,B 0,C 180,E1 -26296.879,E2 -26296.879} C_VEL
LIN {X 0,Y 153.935,Z 515.563,A -85,B 0,C 180,E1 -26300.027,E2 -26300.027} C_VEL
LIN {X 0,Y 155.234,Z 514.834,A -85,B 0,C 180,E1 -26301.237,E2 -26301.237} C_VEL
LIN {X 0,Y 155.717,Z 514.35,A -85,B 0,C 180,E1 -26303.969,E2 -26303.969} C_VEL
LIN {X 0,Y 155.71,Z 514.395,A -85,B 0,C 180,E1 -26306.833,E2 -26306.833} C_VEL
LIN {X 0,Y 155.451,Z 515.013,A -85,B 0,C 180,E1 -26310.817,E2 -26310.817} C_VEL
LIN {X 0,Y 155.094,Z 515.684,A -85,B 0,C 180,E1 -26312.943,E2 -26312.943} C_VEL
LIN {X 0,Y 154.143,Z 517.237,A -85,B 0,C 180,E1 -26316.353,E2 -26316.353} C_VEL
LIN {X 0,Y 152.079,Z 518.908,A -85,B 0,C 180,E1 -26318.24,E2 -26318.24} C_VEL
LIN {X 0,Y 147.93,Z 521.562,A -85,B 0,C 180,E1 -26320.54,E2 -26320.54} C_VEL
LIN {X 0,Y 140.462,Z 525.337,A -85,B 0,C 180,E1 -26323.506,E2 -26323.506} C_VEL
LIN {X 0,Y 133.246,Z 528.32,A -85,B 0,C 180,E1 -26326.728,E2 -26326.728} C_VEL
LIN {X 0,Y 124.677,Z 531.124,A -85,B 0,C 180,E1 -26331.696,E2 -26331.696} C_VEL
LIN {X 0,Y 117.59,Z 532.647,A -85,B 0,C 180,E1 -26337.475,E2 -26337.475} C_VEL
LIN {X 0,Y 111.933,Z 532.922,A -85,B 0,C 180,E1 -26343.943,E2 -26343.943} C_VEL
LIN {X 0,Y 108.067,Z 531.944,A -85,B 0,C 180,E1 -26351.039,E2 -26351.039} C_VEL
LIN {X 0,Y 106.326,Z 529.722,A -85,B 0,C 180,E1 -26358.577,E2 -26358.577} C_VEL
LIN {X 0,Y 106.175,Z 527.665,A -85,B 0,C 180,E1 -26363.188,E2 -26363.188} C_VEL
LIN {X 0,Y 106.429,Z 524.819,A -85,B 0,C 180,E1 -26368.122,E2 -26368.122} C_VEL
LIN {X 0,Y 106.478,Z 521.992,A -85,B 0,C 180,E1 -26371.905,E2 -26371.905} C_VEL
LIN {X 0,Y 106.489,Z 516.6,A -85,B 0,C 180,E1 -26377.599,E2 -26377.599} C_VEL
LIN {X 0,Y 107.144,Z 509.727,A -85,B 0,C 180,E1 -26383.286,E2 -26383.286} C_VEL
LIN {X 0,Y 108.754,Z 501.253,A -85,B 0,C 180,E1 -26388.865,E2 -26388.865} C_VEL
LIN {X 0,Y 110.655,Z 492.579,A -85,B 0,C 180,E1 -26393.402,E2 -26393.402} C_VEL
LIN {X 0,Y 111.925,Z 487.588,A -85,B 0,C 180,E1 -26395.589,E2 -26395.589} C_VEL
LIN {X 0,Y 111.735,Z 476.914,A -85,B 0,C 180,E1 -26399.679,E2 -26399.679} C_VEL
LIN {X 0,Y 111.518,Z 464.934,A -85,B 0,C 180,E1 -26403.48,E2 -26403.48} C_VEL
LIN {X 0,Y 111.142,Z 451.272,A -85,B 0,C 180,E1 -26406.935,E2 -26406.935} C_VEL
LIN {X 0,Y 110.505,Z 437.665,A -85,B 0,C 180,E1 -26409.642,E2 -26409.642} C_VEL
LIN {X 0,Y 109.433,Z 432.428,A -85,B 0,C 180,E1 -26410.644,E2 -26410.644} C_VEL
LIN {X 0,Y 108.989,Z 430.123,A -85,B 0,C 180,E1 -26411.093,E2 -26411.093} C_VEL
LIN {X 0,Y 108.274,Z 427.001,A -85,B 0,C 180,E1 -26417.663,E2 -26417.663} C_VEL
LIN {X 0,Y 107.868,Z 427.043,A -85,B 0,C 180,E1 -26424.095,E2 -26424.095} C_VEL
LIN {X 0,Y 107.83,Z 427.053,A -85,B 0,C 180,E1 -26428.569,E2 -26428.569} C_VEL
LIN {X 0,Y 107.897,Z 427.045,A -85,B 0,C 180,E1 -26436.991,E2 -26436.991} C_VEL
LIN {X 0,Y 107.991,Z 427.033,A -85,B 0,C 180,E1 -26444.908,E2 -26444.908} C_VEL
LIN {X 0,Y 108.248,Z 426.996,A -85,B 0,C 180,E1 -26448.765,E2 -26448.765} C_VEL
LIN {X 0,Y 108.459,Z 426.973,A -85,B 0,C 180,E1 -26456.281,E2 -26456.281} C_VEL
LIN {X 0,Y 108.922,Z 426.914,A -85,B 0,C 180,E1 -26459.997,E2 -26459.997} C_VEL
LIN {X 0,Y 108.306,Z 426.988,A -85,B 0,C 180,E1 -26467.453,E2 -26467.453} C_VEL
LIN {X 0,Y 108.158,Z 427.01,A -85,B 0,C 180,E1 -26472.866,E2 -26472.866} C_VEL
LIN {X 0,Y 107.885,Z 427.047,A -85,B 0,C 180,E1 -26479.005,E2 -26479.005} C_VEL
LIN {X 0,Y 107.902,Z 427.037,A -85,B 0,C 180,E1 -26482.916,E2 -26482.916} C_VEL
LIN {X 0,Y 107.701,Z 427.073,A -85,B 0,C 180,E1 -26484.997,E2 -26484.997} C_VEL
LIN {X 0,Y 106.444,Z 427.242,A -85,B 0,C 180,E1 -26488.088,E2 -26488.088} C_VEL
LIN {X 0,Y 103.219,Z 427.647,A -85,B 0,C 180,E1 -26493.286,E2 -26493.286} C_VEL
LIN {X 0,Y 101.077,Z 427.899,A -85,B 0,C 180,E1 -26497.702,E2 -26497.702} C_VEL
LIN {X 0,Y 100.635,Z 427.941,A -85,B 0,C 180,E1 -26500,E2 -26500} C_VEL
LIN {X 0,Y 100.651,Z 427.946,A -85,B 0,C 180,E1 -26505.694,E2 -26505.694} C_VEL
LIN {X 0,Y 100.631,Z 427.949,A -85,B 0,C 180,E1 -26511.039,E2 -26511.039} C_VEL
LIN {X 0,Y 100.695,Z 427.935,A -85,B 0,C 180,E1 -26516.874,E2 -26516.874} C_VEL
LIN {X 0,Y 100.791,Z 427.922,A -85,B 0,C 180,E1 -26525.253,E2 -26525.253} C_VEL
LIN {X 0,Y 100.819,Z 427.926,A -85,B 0,C 180,E1 -26529.587,E2 -26529.587} C_VEL
LIN {X 0,Y 101.102,Z 427.891,A -85,B 0,C 180,E1 -26536.688,E2 -26536.688} C_VEL
LIN {X 0,Y 101.24,Z 427.867,A -85,B 0,C 180,E1 -26542.005,E2 -26542.005} C_VEL
LIN {X 0,Y 101.86,Z 427.79,A -85,B 0,C 180,E1 -26549.986,E2 -26549.986} C_VEL
LIN {X 0,Y 101.27,Z 427.864,A -85,B 0,C 180,E1 -26557.963,E2 -26557.963} C_VEL
LIN {X 0,Y 101.102,Z 427.891,A -85,B 0,C 180,E1 -26563.312,E2 -26563.312} C_VEL
LIN {X 0,Y 100.817,Z 427.926,A -85,B 0,C 180,E1 -26570.916,E2 -26570.916} C_VEL
LIN {X 0,Y 104.877,Z 441.873,A -85,B 0,C 180,E1 -26574.863,E2 -26574.863} C_VEL
LIN {X 0,Y 107.258,Z 453.132,A -85,B 0,C 180,E1 -26578.346,E2 -26578.346} C_VEL
LIN {X 0,Y 108.483,Z 461.51,A -85,B 0,C 180,E1 -26581.199,E2 -26581.199} C_VEL
LIN {X 0,Y 106.095,Z 471.901,A -85,B 0,C 180,E1 -26584.947,E2 -26584.947} C_VEL
LIN {X 0,Y 103.184,Z 482.932,A -85,B 0,C 180,E1 -26589.987,E2 -26589.987} C_VEL
LIN {X 0,Y 101.16,Z 491.265,A -85,B 0,C 180,E1 -26594.792,E2 -26594.792} C_VEL
LIN {X 0,Y 99.437,Z 499.876,A -85,B 0,C 180,E1 -26601.002,E2 -26601.002} C_VEL
LIN {X 0,Y 98.426,Z 506.879,A -85,B 0,C 180,E1 -26607.381,E2 -26607.381} C_VEL
LIN {X 0,Y 98.213,Z 513.076,A -85,B 0,C 180,E1 -26614.578,E2 -26614.578} C_VEL
LIN {X 0,Y 99.234,Z 517.713,A -85,B 0,C 180,E1 -26621.42,E2 -26621.42} C_VEL
LIN {X 0,Y 101.561,Z 521.227,A -85,B 0,C 180,E1 -26628.022,E2 -26628.022} C_VEL
LIN {X 0,Y 105.759,Z 524.015,A -85,B 0,C 180,E1 -26635.22,E2 -26635.22} C_VEL
LIN {X 0,Y 112.557,Z 525.618,A -85,B 0,C 180,E1 -26642.84,E2 -26642.84} C_VEL
LIN {X 0,Y 117.494,Z 525.781,A -85,B 0,C 180,E1 -26646.874,E2 -26646.874} C_VEL
LIN {X 0,Y 122.055,Z 525.436,A -85,B 0,C 180,E1 -26649.95,E2 -26649.95} C_VEL
LIN {X 0,Y 130.768,Z 523.88,A -85,B 0,C 180,E1 -26654.724,E2 -26654.724} C_VEL
LIN {X 0,Y 141.39,Z 520.694,A -85,B 0,C 180,E1 -26659.229,E2 -26659.229} C_VEL
LIN {X 0,Y 146.632,Z 518.636,A -85,B 0,C 180,E1 -26661.07,E2 -26661.07} C_VEL
LIN {X 0,Y 148.915,Z 517.64,A -85,B 0,C 180,E1 -26662.185,E2 -26662.185} C_VEL
LIN {X 0,Y 149.358,Z 517.399,A -85,B 0,C 180,E1 -26665.058,E2 -26665.058} C_VEL
LIN {X 0,Y 149.213,Z 517.659,A -85,B 0,C 180,E1 -26668.102,E2 -26668.102} C_VEL
LIN {X 0,Y 148.832,Z 518.422,A -85,B 0,C 180,E1 -26671.813,E2 -26671.813} C_VEL
LIN {X 0,Y 148.125,Z 519.448,A -85,B 0,C 180,E1 -26674.708,E2 -26674.708} C_VEL
LIN {X 0,Y 147.389,Z 520.101,A -85,B 0,C 180,E1 -26675.864,E2 -26675.864} C_VEL
LIN {X 0,Y 145.575,Z 521.257,A -85,B 0,C 180,E1 -26677.214,E2 -26677.214} C_VEL
LIN {X 0,Y 143.388,Z 522.492,A -85,B 0,C 180,E1 -26678.37,E2 -26678.37} C_VEL
LIN {X 0,Y 138.285,Z 524.829,A -85,B 0,C 180,E1 -26680.348,E2 -26680.348} C_VEL
LIN {X 0,Y 128.189,Z 528.59,A -85,B 0,C 180,E1 -26684.561,E2 -26684.561} C_VEL
LIN {X 0,Y 119.187,Z 531.057,A -85,B 0,C 180,E1 -26689.58,E2 -26689.58} C_VEL
LIN {X 0,Y 111.652,Z 532.295,A -85,B 0,C 180,E1 -26695.51,E2 -26695.51} C_VEL
LIN {X 0,Y 105.594,Z 532.294,A -85,B 0,C 180,E1 -26702.248,E2 -26702.248} C_VEL
LIN {X 0,Y 101.392,Z 531.027,A -85,B 0,C 180,E1 -26709.738,E2 -26709.738} C_VEL
LIN {X 0,Y 99.443,Z 528.508,A -85,B 0,C 180,E1 -26717.775,E2 -26717.775} C_VEL
LIN {X 0,Y 99.227,Z 526.414,A -85,B 0,C 180,E1 -26722.586,E2 -26722.586} C_VEL
LIN {X 0,Y 99.5,Z 523.298,A -85,B 0,C 180,E1 -26727.991,E2 -26727.991} C_VEL
LIN {X 0,Y 99.521,Z 520.293,A -85,B 0,C 180,E1 -26732.038,E2 -26732.038} C_VEL
LIN {X 0,Y 99.576,Z 514.616,A -85,B 0,C 180,E1 -26738.13,E2 -26738.13} C_VEL
LIN {X 0,Y 100.312,Z 507.474,A -85,B 0,C 180,E1 -26744.209,E2 -26744.209} C_VEL
LIN {X 0,Y 101.752,Z 500.251,A -85,B 0,C 180,E1 -26749.167,E2 -26749.167} C_VEL
LIN {X 0,Y 103.742,Z 491.45,A -85,B 0,C 180,E1 -26753.998,E2 -26753.998} C_VEL
LIN {X 0,Y 104.81,Z 487.477,A -85,B 0,C 180,E1 -26755.854,E2 -26755.854} C_VEL
LIN {X 0,Y 104.686,Z 476.843,A -85,B 0,C 180,E1 -26760.23,E2 -26760.23} C_VEL
LIN {X 0,Y 104.535,Z 465.301,A -85,B 0,C 180,E1 -26764.177,E2 -26764.177} C_VEL
LIN {X 0,Y 104.328,Z 453.032,A -85,B 0,C 180,E1 -26767.583,E2 -26767.583} C_VEL
LIN {X 0,Y 103.792,Z 438.973,A -85,B 0,C 180,E1 -26770.653,E2 -26770.653} C_VEL
LIN {X 0,Y 102.396,Z 432.464,A -85,B 0,C 180,E1 -26772.023,E2 -26772.023} C_VEL
LIN {X 0,Y 101.7,Z 429.712,A -85,B 0,C 180,E1 -26772.632,E2 -26772.632} C_VEL
LIN {X 0,Y 101.264,Z 427.874,A -85,B 0,C 180,E1 -26777.14,E2 -26777.14} C_VEL
LIN {X 0,Y 100.999,Z 427.905,A -85,B 0,C 180,E1 -26781.221,E2 -26781.221} C_VEL
LIN {X 0,Y 100.742,Z 427.932,A -85,B 0,C 180,E1 -26786.864,E2 -26786.864} C_VEL
LIN {X 0,Y 100.766,Z 427.93,A -85,B 0,C 180,E1 -26795.258,E2 -26795.258} C_VEL
LIN {X 0,Y 100.802,Z 427.926,A -85,B 0,C 180,E1 -26799.594,E2 -26799.594} C_VEL
LIN {X 0,Y 101.147,Z 427.883,A -85,B 0,C 180,E1 -26807.965,E2 -26807.965} C_VEL
LIN {X 0,Y 101.253,Z 427.87,A -85,B 0,C 180,E1 -26812.017,E2 -26812.017} C_VEL
LIN {X 0,Y 101.849,Z 427.794,A -85,B 0,C 180,E1 -26819.996,E2 -26819.996} C_VEL
LIN {X 0,Y 101.241,Z 427.869,A -85,B 0,C 180,E1 -26827.977,E2 -26827.977} C_VEL
LIN {X 0,Y 101.07,Z 427.892,A -85,B 0,C 180,E1 -26833.164,E2 -26833.164} C_VEL
LIN {X 0,Y 100.806,Z 427.928,A -85,B 0,C 180,E1 -26840.397,E2 -26840.397} C_VEL
LIN {X 0,Y 100.759,Z 427.929,A -85,B 0,C 180,E1 -26844.908,E2 -26844.908} C_VEL
LIN {X 0,Y 100.704,Z 427.936,A -85,B 0,C 180,E1 -26853.102,E2 -26853.102} C_VEL
LIN {X 0,Y 100.635,Z 427.941,A -85,B 0,C 180,E1 -26860,E2 -26860} C_VEL
LIN {X 0,Y 99.871,Z 428.044,A -85,B 0,C 180,E1 -26863.344,E2 -26863.344} C_VEL
LIN {X 0,Y 98.345,Z 428.235,A -85,B 0,C 180,E1 -26866.662,E2 -26866.662} C_VEL
LIN {X 0,Y 93.983,Z 428.786,A -85,B 0,C 180,E1 -26875.914,E2 -26875.914} C_VEL
LIN {X 0,Y 93.579,Z 428.822,A -85,B 0,C 180,E1 -26878.371,E2 -26878.371} C_VEL
LIN {X 0,Y 93.673,Z 428.81,A -85,B 0,C 180,E1 -26884.191,E2 -26884.191} C_VEL
LIN {X 0,Y 93.697,Z 428.812,A -85,B 0,C 180,E1 -26887.957,E2 -26887.957} C_VEL
LIN {X 0,Y 94.022,Z 428.772,A -85,B 0,C 180,E1 -26896.326,E2 -26896.326} C_VEL
LIN {X 0,Y 94.173,Z 428.748,A -85,B 0,C 180,E1 -26901.401,E2 -26901.401} C_VEL
LIN {X 0,Y 94.786,Z 428.671,A -85,B 0,C 180,E1 -26909.984,E2 -26909.984} C_VEL
LIN {X 0,Y 94.201,Z 428.743,A -85,B 0,C 180,E1 -26918.565,E2 -26918.565} C_VEL
LIN {X 0,Y 94.018,Z 428.774,A -85,B 0,C 180,E1 -26923.665,E2 -26923.665} C_VEL
LIN {X 0,Y 93.74,Z 428.806,A -85,B 0,C 180,E1 -26929.415,E2 -26929.415} C_VEL
LIN {X 0,Y 97.536,Z 441.319,A -85,B 0,C 180,E1 -26933.33,E2 -26933.33} C_VEL
LIN {X 0,Y 100.102,Z 452.744,A -85,B 0,C 180,E1 -26937.135,E2 -26937.135} C_VEL
LIN {X 0,Y 101.418,Z 462.6,A -85,B 0,C 180,E1 -26940.746,E2 -26940.746} C_VEL
LIN {X 0,Y 98.865,Z 472.66,A -85,B 0,C 180,E1 -26944.64,E2 -26944.64} C_VEL
LIN {X 0,Y 95.732,Z 484.083,A -85,B 0,C 180,E1 -26950.288,E2 -26950.288} C_VEL
LIN {X 0,Y 93.581,Z 493.035,A -85,B 0,C 180,E1 -26956.004,E2 -26956.004} C_VEL
LIN {X 0,Y 92.102,Z 500.958,A -85,B 0,C 180,E1 -26962.383,E2 -26962.383} C_VEL
LIN {X 0,Y 91.256,Z 507.479,A -85,B 0,C 180,E1 -26968.956,E2 -26968.956} C_VEL
LIN {X 0,Y 91.417,Z 514.125,A -85,B 0,C 180,E1 -26977.398,E2 -26977.398} C_VEL
LIN {X 0,Y 93.003,Z 518.622,A -85,B 0,C 180,E1 -26984.67,E2 -26984.67} C_VEL
LIN {X 0,Y 95.962,Z 521.987,A -85,B 0,C 180,E1 -26991.581,E2 -26991.581} C_VEL
LIN {X 0,Y 98.613,Z 523.66,A -85,B 0,C 180,E1 -26995.917,E2 -26995.917} C_VEL
LIN {X 0,Y 105.475,Z 525.793,A -85,B 0,C 180,E1 -27003.824,E2 -27003.824} C_VEL
LIN {X 0,Y 109.656,Z 526.264,A -85,B 0,C 180,E1 -27007.368,E2 -27007.368} C_VEL
LIN {X 0,Y 119.269,Z 525.918,A -85,B 0,C 180,E1 -27013.636,E2 -27013.636} C_VEL
LIN {X 0,Y 124.633,Z 525.149,A -85,B 0,C 180,E1 -27016.379,E2 -27016.379} C_VEL
LIN {X 0,Y 135.343,Z 522.587,A -85,B 0,C 180,E1 -27020.857,E2 -27020.857} C_VEL
LIN {X 0,Y 142.363,Z 520.227,A -85,B 0,C 180,E1 -27023.264,E2 -27023.264} C_VEL
LIN {X 0,Y 142.786,Z 520.225,A -85,B 0,C 180,E1 -27026.297,E2 -27026.297} C_VEL
LIN {X 0,Y 142.466,Z 520.678,A -85,B 0,C 180,E1 -27029.561,E2 -27029.561} C_VEL
LIN {X 0,Y 141.878,Z 521.556,A -85,B 0,C 180,E1 -27033.02,E2 -27033.02} C_VEL
LIN {X 0,Y 140.973,Z 522.29,A -85,B 0,C 180,E1 -27034.85,E2 -27034.85} C_VEL
LIN {X 0,Y 139.027,Z 523.278,A -85,B 0,C 180,E1 -27036.04,E2 -27036.04} C_VEL
LIN {X 0,Y 136.549,Z 524.372,A -85,B 0,C 180,E1 -27037.103,E2 -27037.103} C_VEL
LIN {X 0,Y 128.471,Z 527.303,A -85,B 0,C 180,E1 -27040.036,E2 -27040.036} C_VEL
LIN {X 0,Y 118.42,Z 530.042,A -85,B 0,C 180,E1 -27044.607,E2 -27044.607} C_VEL
LIN {X 0,Y 109.652,Z 531.544,A -85,B 0,C 180,E1 -27050.157,E2 -27050.157} C_VEL
LIN {X 0,Y 102.385,Z 531.845,A -85,B 0,C 180,E1 -27056.71,E2 -27056.71} C_VEL
LIN {X 0,Y 96.793,Z 530.925,A -85,B 0,C 180,E1 -27064.191,E2 -27064.191} C_VEL
LIN {X 0,Y 93.437,Z 528.814,A -85,B 0,C 180,E1 -27072.507,E2 -27072.507} C_VEL
LIN {X 0,Y 92.303,Z 525.349,A -85,B 0,C 180,E1 -27081.257,E2 -27081.257} C_VEL
LIN {X 0,Y 92.58,Z 521.725,A -85,B 0,C 180,E1 -27087.841,E2 -27087.841} C_VEL
LIN {X 0,Y 92.559,Z 518.55,A -85,B 0,C 180,E1 -27092.192,E2 -27092.192} C_VEL
LIN {X 0,Y 92.644,Z 512.537,A -85,B 0,C 180,E1 -27098.742,E2 -27098.742} C_VEL
LIN {X 0,Y 93.566,Z 505.001,A -85,B 0,C 180,E1 -27105.258,E2 -27105.258} C_VEL
LIN {X 0,Y 95.125,Z 497.368,A -85,B 0,C 180,E1 -27110.561,E2 -27110.561} C_VEL
LIN {X 0,Y 97.706,Z 487.209,A -85,B 0,C 180,E1 -27116.156,E2 -27116.156} C_VEL
LIN {X 0,Y 97.624,Z 476.519,A -85,B 0,C 180,E1 -27120.876,E2 -27120.876} C_VEL
LIN {X 0,Y 97.543,Z 464.635,A -85,B 0,C 180,E1 -27125.215,E2 -27125.215} C_VEL
LIN {X 0,Y 97.417,Z 452.778,A -85,B 0,C 180,E1 -27128.731,E2 -27128.731} C_VEL
LIN {X 0,Y 96.914,Z 439.083,A -85,B 0,C 180,E1 -27131.982,E2 -27131.982} C_VEL
LIN {X 0,Y 94.927,Z 431.745,A -85,B 0,C 180,E1 -27133.788,E2 -27133.788} C_VEL
LIN {X 0,Y 94.384,Z 429.298,A -85,B 0,C 180,E1 -27134.404,E2 -27134.404} C_VEL
LIN {X 0,Y 94.231,Z 428.75,A -85,B 0,C 180,E1 -27136.374,E2 -27136.374} C_VEL
LIN {X 0,Y 94.177,Z 428.755,A -85,B 0,C 180,E1 -27138.289,E2 -27138.289} C_VEL
LIN {X 0,Y 93.69,Z 428.808,A -85,B 0,C 180,E1 -27145.629,E2 -27145.629} C_VEL
LIN {X 0,Y 93.666,Z 428.812,A -85,B 0,C 180,E1 -27154.241,E2 -27154.241} C_VEL
LIN {X 0,Y 93.677,Z 428.816,A -85,B 0,C 180,E1 -27157.964,E2 -27157.964} C_VEL
LIN {X 0,Y 94.039,Z 428.77,A -85,B 0,C 180,E1 -27167.04,E2 -27167.04} C_VEL
LIN {X 0,Y 94.183,Z 428.748,A -85,B 0,C 180,E1 -27171.413,E2 -27171.413} C_VEL
LIN {X 0,Y 94.778,Z 428.675,A -85,B 0,C 180,E1 -27179.996,E2 -27179.996} C_VEL
LIN {X 0,Y 94.152,Z 428.753,A -85,B 0,C 180,E1 -27188.582,E2 -27188.582} C_VEL
LIN {X 0,Y 93.979,Z 428.775,A -85,B 0,C 180,E1 -27193.488,E2 -27193.488} C_VEL
LIN {X 0,Y 93.679,Z 428.812,A -85,B 0,C 180,E1 -27202.027,E2 -27202.027} C_VEL
LIN {X 0,Y 93.622,Z 428.823,A -85,B 0,C 180,E1 -27206.765,E2 -27206.765} C_VEL
LIN {X 0,Y 93.6,Z 428.824,A -85,B 0,C 180,E1 -27214.291,E2 -27214.291} C_VEL
LIN {X 0,Y 93.54,Z 428.831,A -85,B 0,C 180,E1 -27222.542,E2 -27222.542} C_VEL
LIN {X 0,Y 93.541,Z 428.826,A -85,B 0,C 180,E1 -27228.7,E2 -27228.7} C_VEL
LIN {X 0,Y 93.592,Z 428.822,A -85,B 0,C 180,E1 -27235.684,E2 -27235.684} C_VEL
LIN {X 0,Y 93.579,Z 428.822,A -85,B 0,C 180,E1 -27238.371,E2 -27238.371} C_VEL
LIN {X 0,Y 92.796,Z 428.926,A -85,B 0,C 180,E1 -27241.968,E2 -27241.968} C_VEL
LIN {X 0,Y 91.256,Z 429.116,A -85,B 0,C 180,E1 -27245.543,E2 -27245.543} C_VEL
LIN {X 0,Y 87.143,Z 429.627,A -85,B 0,C 180,E1 -27255.569,E2 -27255.569} C_VEL
LIN {X 0,Y 86.929,Z 429.643,A -85,B 0,C 180,E1 -27258.225,E2 -27258.225} C_VEL
LIN {X 0,Y 87.083,Z 429.632,A -85,B 0,C 180,E1 -27260.694,E2 -27260.694} C_VEL
LIN {X 0,Y 87.712,Z 429.552,A -85,B 0,C 180,E1 -27269.983,E2 -27269.983} C_VEL
LIN {X 0,Y 87.105,Z 429.627,A -85,B 0,C 180,E1 -27279.269,E2 -27279.269} C_VEL
LIN {X 0,Y 86.764,Z 429.669,A -85,B 0,C 180,E1 -27286.451,E2 -27286.451} C_VEL
LIN {X 0,Y 86.736,Z 429.673,A -85,B 0,C 180,E1 -27287.823,E2 -27287.823} C_VEL
LIN {X 0,Y 90.273,Z 441.059,A -85,B 0,C 180,E1 -27291.685,E2 -27291.685} C_VEL
LIN {X 0,Y 92.617,Z 451.048,A -85,B 0,C 180,E1 -27295.249,E2 -27295.249} C_VEL
LIN {X 0,Y 94.18,Z 460.652,A -85,B 0,C 180,E1 -27298.997,E2 -27298.997} C_VEL
LIN {X 0,Y 94.21,Z 463.702,A -85,B 0,C 180,E1 -27300.215,E2 -27300.215} C_VEL
LIN {X 0,Y 91.145,Z 474.933,A -85,B 0,C 180,E1 -27304.995,E2 -27304.995} C_VEL
LIN {X 0,Y 88.489,Z 484.441,A -85,B 0,C 180,E1 -27310.207,E2 -27310.207} C_VEL
LIN {X 0,Y 86.239,Z 493.756,A -85,B 0,C 180,E1 -27316.742,E2 -27316.742} C_VEL
LIN {X 0,Y 84.737,Z 502.433,A -85,B 0,C 180,E1 -27324.515,E2 -27324.515} C_VEL
LIN {X 0,Y 84.089,Z 509.54,A -85,B 0,C 180,E1 -27332.639,E2 -27332.639} C_VEL
LIN {X 0,Y 84.81,Z 515.067,A -85,B 0,C 180,E1 -27340.647,E2 -27340.647} C_VEL
LIN {X 0,Y 86.545,Z 518.67,A -85,B 0,C 180,E1 -27346.942,E2 -27346.942} C_VEL
LIN {X 0,Y 90.763,Z 522.705,A -85,B 0,C 180,E1 -27355.563,E2 -27355.563} C_VEL
LIN {X 0,Y 97.619,Z 525.541,A -85,B 0,C 180,E1 -27364.132,E2 -27364.132} C_VEL
LIN {X 0,Y 101.813,Z 526.383,A -85,B 0,C 180,E1 -27367.939,E2 -27367.939} C_VEL
LIN {X 0,Y 107.888,Z 526.834,A -85,B 0,C 180,E1 -27372.352,E2 -27372.352} C_VEL
LIN {X 0,Y 118.23,Z 526.304,A -85,B 0,C 180,E1 -27378.038,E2 -27378.038} C_VEL
LIN {X 0,Y 129.419,Z 524.26,A -85,B 0,C 180,E1 -27382.64,E2 -27382.64} C_VEL
LIN {X 0,Y 135.193,Z 522.728,A -85,B 0,C 180,E1 -27384.578,E2 -27384.578} C_VEL
LIN {X 0,Y 135.979,Z 522.755,A -85,B 0,C 180,E1 -27387.723,E2 -27387.723} C_VEL
LIN {X 0,Y 135.402,Z 523.435,A -85,B 0,C 180,E1 -27391.271,E2 -27391.271} C_VEL
LIN {X 0,Y 134.739,Z 524.049,A -85,B 0,C 180,E1 -27393.452,E2 -27393.452} C_VEL
LIN {X 0,Y 129.592,Z 525.93,A -85,B 0,C 180,E1 -27395.585,E2 -27395.585} C_VEL
LIN {X 0,Y 118.674,Z 528.963,A -85,B 0,C 180,E1 -27399.679,E2 -27399.679} C_VEL
LIN {X 0,Y 108.772,Z 530.75,A -85,B 0,C 180,E1 -27404.727,E2 -27404.727} C_VEL
LIN {X 0,Y 100.242,Z 531.354,A -85,B 0,C 180,E1 -27410.897,E2 -27410.897} C_VEL
LIN {X 0,Y 93.31,Z 530.762,A -85,B 0,C 180,E1 -27418.201,E2 -27418.201} C_VEL
LIN {X 0,Y 88.308,Z 528.926,A -85,B 0,C 180,E1 -27426.57,E2 -27426.57} C_VEL
LIN {X 0,Y 85.808,Z 525.892,A -85,B 0,C 180,E1 -27435.794,E2 -27435.794} C_VEL
LIN {X 0,Y 85.565,Z 521.402,A -85,B 0,C 180,E1 -27445.306,E2 -27445.306} C_VEL
LIN {X 0,Y 85.658,Z 518.41,A -85,B 0,C 180,E1 -27450.017,E2 -27450.017} C_VEL
LIN {X 0,Y 85.612,Z 512.622,A -85,B 0,C 180,E1 -27457.09,E2 -27457.09} C_VEL
LIN {X 0,Y 86.314,Z 505.271,A -85,B 0,C 180,E1 -27464.156,E2 -27464.156} C_VEL
LIN {X 0,Y 87.814,Z 497.806,A -85,B 0,C 180,E1 -27469.902,E2 -27469.902} C_VEL
LIN {X 0,Y 90.019,Z 488.793,A -85,B 0,C 180,E1 -27475.447,E2 -27475.447} C_VEL
LIN {X 0,Y 90.703,Z 485.663,A -85,B 0,C 180,E1 -27477.096,E2 -27477.096} C_VEL
LIN {X 0,Y 90.607,Z 474.239,A -85,B 0,C 180,E1 -27482.422,E2 -27482.422} C_VEL
LIN {X 0,Y 90.564,Z 462.24,A -85,B 0,C 180,E1 -27486.991,E2 -27486.991} C_VEL
LIN {X 0,Y 90.488,Z 449.812,A -85,B 0,C 180,E1 -27490.816,E2 -27490.816} C_VEL
LIN {X 0,Y 90.229,Z 440.676,A -85,B 0,C 180,E1 -27493.152,E2 -27493.152} C_VEL
LIN {X 0,Y 87.948,Z 432.079,A -85,B 0,C 180,E1 -27495.508,E2 -27495.508} C_VEL
LIN {X 0,Y 87.208,Z 429.624,A -85,B 0,C 180,E1 -27496.21,E2 -27496.21} C_VEL
LIN {X 0,Y 86.659,Z 429.683,A -85,B 0,C 180,E1 -27505.406,E2 -27505.406} C_VEL
LIN {X 0,Y 86.589,Z 429.691,A -85,B 0,C 180,E1 -27513.263,E2 -27513.263} C_VEL
LIN {X 0,Y 86.621,Z 429.688,A -85,B 0,C 180,E1 -27521.058,E2 -27521.058} C_VEL
LIN {X 0,Y 86.886,Z 429.662,A -85,B 0,C 180,E1 -27526.149,E2 -27526.149} C_VEL
LIN {X 0,Y 87.07,Z 429.631,A -85,B 0,C 180,E1 -27530.706,E2 -27530.706} C_VEL
LIN {X 0,Y 87.708,Z 429.556,A -85,B 0,C 180,E1 -27539.996,E2 -27539.996} C_VEL
LIN {X 0,Y 87.046,Z 429.641,A -85,B 0,C 180,E1 -27549.288,E2 -27549.288} C_VEL
LIN {X 0,Y 86.88,Z 429.657,A -85,B 0,C 180,E1 -27554.04,E2 -27554.04} C_VEL
LIN {X 0,Y 86.622,Z 429.696,A -85,B 0,C 180,E1 -27558.933,E2 -27558.933} C_VEL
LIN {X 0,Y 86.587,Z 429.699,A -85,B 0,C 180,E1 -27566.734,E2 -27566.734} C_VEL
LIN {X 0,Y 86.518,Z 429.708,A -85,B 0,C 180,E1 -27575.65,E2 -27575.65} C_VEL
LIN {X 0,Y 86.484,Z 429.711,A -85,B 0,C 180,E1 -27582.975,E2 -27582.975} C_VEL
LIN {X 0,Y 86.463,Z 429.708,A -85,B 0,C 180,E1 -27589.417,E2 -27589.417} C_VEL
LIN {X 0,Y 86.535,Z 429.702,A -85,B 0,C 180,E1 -27595.334,E2 -27595.334} C_VEL
LIN {X 0,Y 86.588,Z 429.696,A -85,B 0,C 180,E1 -27603.22,E2 -27603.22} C_VEL
LIN {X 0,Y 86.648,Z 429.69,A -85,B 0,C 180,E1 -27611.051,E2 -27611.051} C_VEL
LIN {X 0,Y 86.931,Z 429.654,A -85,B 0,C 180,E1 -27615.947,E2 -27615.947} C_VEL
LIN {X 0,Y 86.929,Z 429.643,A -85,B 0,C 180,E1 -27618.225,E2 -27618.225} C_VEL
LIN {X 0,Y 86.668,Z 429.684,A -85,B 0,C 180,E1 -27620.814,E2 -27620.814} C_VEL
LIN {X 0,Y 85.355,Z 429.852,A -85,B 0,C 180,E1 -27624.665,E2 -27624.665} C_VEL
LIN {X 0,Y 82.169,Z 430.248,A -85,B 0,C 180,E1 -27631.208,E2 -27631.208} C_VEL
LIN {X 0,Y 80.231,Z 430.488,A -85,B 0,C 180,E1 -27636.827,E2 -27636.827} C_VEL
LIN {X 0,Y 79.969,Z 430.516,A -85,B 0,C 180,E1 -27639.745,E2 -27639.745} C_VEL
LIN {X 0,Y 79.74,Z 430.553,A -85,B 0,C 180,E1 -27645.968,E2 -27645.968} C_VEL
LIN {X 0,Y 83.347,Z 442.108,A -85,B 0,C 180,E1 -27650.335,E2 -27650.335} C_VEL
LIN {X 0,Y 85.659,Z 451.907,A -85,B 0,C 180,E1 -27654.2,E2 -27654.2} C_VEL
LIN {X 0,Y 87.052,Z 460.384,A -85,B 0,C 180,E1 -27657.769,E2 -27657.769} C_VEL
LIN {X 0,Y 87.378,Z 462.82,A -85,B 0,C 180,E1 -27658.835,E2 -27658.835} C_VEL
LIN {X 0,Y 84.854,Z 472.3,A -85,B 0,C 180,E1 -27663.016,E2 -27663.016} C_VEL
LIN {X 0,Y 81.638,Z 483.263,A -85,B 0,C 180,E1 -27669.222,E2 -27669.222} C_VEL
LIN {X 0,Y 79.177,Z 493.2,A -85,B 0,C 180,E1 -27676.542,E2 -27676.542} C_VEL
LIN {X 0,Y 77.715,Z 501.515,A -85,B 0,C 180,E1 -27684.444,E2 -27684.444} C_VEL
LIN {X 0,Y 77.086,Z 508.467,A -85,B 0,C 180,E1 -27692.885,E2 -27692.885} C_VEL
LIN {X 0,Y 77.904,Z 514.276,A -85,B 0,C 180,E1 -27701.599,E2 -27701.599} C_VEL
LIN {X 0,Y 80.394,Z 518.897,A -85,B 0,C 180,E1 -27709.935,E2 -27709.935} C_VEL
LIN {X 0,Y 84.381,Z 522.397,A -85,B 0,C 180,E1 -27717.609,E2 -27717.609} C_VEL
LIN {X 0,Y 91.979,Z 525.666,A -85,B 0,C 180,E1 -27726.783,E2 -27726.783} C_VEL
LIN {X 0,Y 101.463,Z 527.205,A -85,B 0,C 180,E1 -27734.199,E2 -27734.199} C_VEL
LIN {X 0,Y 112.153,Z 527.22,A -85,B 0,C 180,E1 -27739.998,E2 -27739.998} C_VEL
LIN {X 0,Y 123.649,Z 525.75,A -85,B 0,C 180,E1 -27744.609,E2 -27744.609} C_VEL
LIN {X 0,Y 128.01,Z 524.878,A -85,B 0,C 180,E1 -27746.057,E2 -27746.057} C_VEL
LIN {X 0,Y 128.822,Z 525.031,A -85,B 0,C 180,E1 -27749.409,E2 -27749.409} C_VEL
LIN {X 0,Y 128.172,Z 525.592,A -85,B 0,C 180,E1 -27751.907,E2 -27751.907} C_VEL
LIN {X 0,Y 125.574,Z 526.408,A -85,B 0,C 180,E1 -27752.937,E2 -27752.937} C_VEL
LIN {X 0,Y 114.272,Z 529.027,A -85,B 0,C 180,E1 -27756.939,E2 -27756.939} C_VEL
LIN {X 0,Y 103.896,Z 530.462,A -85,B 0,C 180,E1 -27761.942,E2 -27761.942} C_VEL
LIN {X 0,Y 94.844,Z 530.734,A -85,B 0,C 180,E1 -27768.194,E2 -27768.194} C_VEL
LIN {X 0,Y 87.378,Z 529.835,A -85,B 0,C 180,E1 -27775.757,E2 -27775.757} C_VEL
LIN {X 0,Y 81.898,Z 527.761,A -85,B 0,C 180,E1 -27784.612,E2 -27784.612} C_VEL
LIN {X 0,Y 79.056,Z 524.438,A -85,B 0,C 180,E1 -27794.552,E2 -27794.552} C_VEL
LIN {X 0,Y 78.578,Z 521.214,A -85,B 0,C 180,E1 -27801.917,E2 -27801.917} C_VEL
LIN {X 0,Y 78.808,Z 518.204,A -85,B 0,C 180,E1 -27807.463,E2 -27807.463} C_VEL
LIN {X 0,Y 78.688,Z 513.611,A -85,B 0,C 180,E1 -27813.86,E2 -27813.86} C_VEL
LIN {X 0,Y 79.027,Z 506.32,A -85,B 0,C 180,E1 -27821.953,E2 -27821.953} C_VEL
LIN {X 0,Y 80.533,Z 498.131,A -85,B 0,C 180,E1 -27829.121,E2 -27829.121} C_VEL
LIN {X 0,Y 83.201,Z 487.412,A -85,B 0,C 180,E1 -27836.344,E2 -27836.344} C_VEL
LIN {X 0,Y 83.562,Z 483.995,A -85,B 0,C 180,E1 -27838.254,E2 -27838.254} C_VEL
LIN {X 0,Y 83.583,Z 473.032,A -85,B 0,C 180,E1 -27843.699,E2 -27843.699} C_VEL
LIN {X 0,Y 83.657,Z 460.634,A -85,B 0,C 180,E1 -27848.69,E2 -27848.69} C_VEL
LIN {X 0,Y 83.702,Z 448.307,A -85,B 0,C 180,E1 -27852.703,E2 -27852.703} C_VEL
LIN {X 0,Y 83.652,Z 442.88,A -85,B 0,C 180,E1 -27854.202,E2 -27854.202} C_VEL
LIN {X 0,Y 81.495,Z 434.45,A -85,B 0,C 180,E1 -27856.796,E2 -27856.796} C_VEL
LIN {X 0,Y 79.968,Z 430.524,A -85,B 0,C 180,E1 -27858.129,E2 -27858.129} C_VEL
LIN {X 0,Y 79.658,Z 430.561,A -85,B 0,C 180,E1 -27862.593,E2 -27862.593} C_VEL
LIN {X 0,Y 79.493,Z 430.577,A -85,B 0,C 180,E1 -27872.177,E2 -27872.177} C_VEL
LIN {X 0,Y 79.5,Z 430.58,A -85,B 0,C 180,E1 -27879.287,E2 -27879.287} C_VEL
LIN {X 0,Y 79.81,Z 430.544,A -85,B 0,C 180,E1 -27885.683,E2 -27885.683} C_VEL
LIN {X 0,Y 79.949,Z 430.518,A -85,B 0,C 180,E1 -27889.87,E2 -27889.87} C_VEL
LIN {X 0,Y 80.637,Z 430.436,A -85,B 0,C 180,E1 -27899.996,E2 -27899.996} C_VEL
LIN {X 0,Y 79.931,Z 430.528,A -85,B 0,C 180,E1 -27910.124,E2 -27910.124} C_VEL
LIN {X 0,Y 79.709,Z 430.548,A -85,B 0,C 180,E1 -27915.333,E2 -27915.333} C_VEL
LIN {X 0,Y 79.5,Z 430.581,A -85,B 0,C 180,E1 -27920.703,E2 -27920.703} C_VEL
LIN {X 0,Y 79.487,Z 430.584,A -85,B 0,C 180,E1 -27927.814,E2 -27927.814} C_VEL
LIN {X 0,Y 79.388,Z 430.588,A -85,B 0,C 180,E1 -27932.079,E2 -27932.079} C_VEL
LIN {X 0,Y 79.377,Z 430.594,A -85,B 0,C 180,E1 -27938.294,E2 -27938.294} C_VEL
LIN {X 0,Y 79.396,Z 430.595,A -85,B 0,C 180,E1 -27945.077,E2 -27945.077} C_VEL
LIN {X 0,Y 79.392,Z 430.596,A -85,B 0,C 180,E1 -27952.809,E2 -27952.809} C_VEL
LIN {X 0,Y 79.486,Z 430.583,A -85,B 0,C 180,E1 -27962.141,E2 -27962.141} C_VEL
LIN {X 0,Y 79.516,Z 430.58,A -85,B 0,C 180,E1 -27969.277,E2 -27969.277} C_VEL
LIN {X 0,Y 79.825,Z 430.538,A -85,B 0,C 180,E1 -27975.554,E2 -27975.554} C_VEL
LIN {X 0,Y 79.966,Z 430.521,A -85,B 0,C 180,E1 -27979.858,E2 -27979.858} C_VEL
LIN {X 0,Y 80.639,Z 430.433,A -85,B 0,C 180,E1 -27989.982,E2 -27989.982} C_VEL
LIN {X 0,Y 79.969,Z 430.516,A -85,B 0,C 180,E1 -27999.745,E2 -27999.745} C_VEL
LIN {X 0,Y 79.933,Z 431.198,A -85,B 0,C 180,E1 -28002.014,E2 -28002.014} C_VEL
LIN {X 0,Y 79.723,Z 433.453,A -85,B 0,C 180,E1 -28004.577,E2 -28004.577} C_VEL
LIN {X 0,Y 79.299,Z 437.894,A -85,B 0,C 180,E1 -28007.364,E2 -28007.364} C_VEL
LIN {X 0,Y 78.833,Z 443.709,A -85,B 0,C 180,E1 -28009.624,E2 -28009.624} C_VEL
LIN {X 0,Y 78.706,Z 451.528,A -85,B 0,C 180,E1 -28012.47,E2 -28012.47} C_VEL
LIN {X 0,Y 79.156,Z 455.143,A -85,B 0,C 180,E1 -28014.067,E2 -28014.067} C_VEL
LIN {X 0,Y 80.347,Z 463.302,A -85,B 0,C 180,E1 -28017.918,E2 -28017.918} C_VEL
LIN {X 0,Y 77.634,Z 472.833,A -85,B 0,C 180,E1 -28022.47,E2 -28022.47} C_VEL
LIN {X 0,Y 74.186,Z 484.378,A -85,B 0,C 180,E1 -28029.679,E2 -28029.679} C_VEL
LIN {X 0,Y 71.978,Z 493.171,A -85,B 0,C 180,E1 -28036.89,E2 -28036.89} C_VEL
LIN {X 0,Y 70.582,Z 501.053,A -85,B 0,C 180,E1 -28045.079,E2 -28045.079} C_VEL
LIN {X 0,Y 70.105,Z 508.166,A -85,B 0,C 180,E1 -28054.402,E2 -28054.402} C_VEL
LIN {X 0,Y 71.605,Z 514.814,A -85,B 0,C 180,E1 -28065.185,E2 -28065.185} C_VEL
LIN {X 0,Y 75.069,Z 519.633,A -85,B 0,C 180,E1 -28074.633,E2 -28074.633} C_VEL
LIN {X 0,Y 78.144,Z 522.053,A -85,B 0,C 180,E1 -28080.005,E2 -28080.005} C_VEL
LIN {X 0,Y 85.251,Z 525.286,A -85,B 0,C 180,E1 -28088.531,E2 -28088.531} C_VEL
LIN {X 0,Y 95.159,Z 527.389,A -85,B 0,C 180,E1 -28096.297,E2 -28096.297} C_VEL
LIN {X 0,Y 106.253,Z 527.929,A -85,B 0,C 180,E1 -28102.22,E2 -28102.22} C_VEL
LIN {X 0,Y 118.084,Z 527.021,A -85,B 0,C 180,E1 -28106.81,E2 -28106.81} C_VEL
LIN {X 0,Y 120.893,Z 526.644,A -85,B 0,C 180,E1 -28107.718,E2 -28107.718} C_VEL
LIN {X 0,Y 121.661,Z 526.762,A -85,B 0,C 180,E1 -28109.973,E2 -28109.973} C_VEL
LIN {X 0,Y 115.95,Z 528.035,A -85,B 0,C 180,E1 -28111.97,E2 -28111.97} C_VEL
LIN {X 0,Y 104.58,Z 529.717,A -85,B 0,C 180,E1 -28116.278,E2 -28116.278} C_VEL
LIN {X 0,Y 94.283,Z 530.227,A -85,B 0,C 180,E1 -28121.831,E2 -28121.831} C_VEL
LIN {X 0,Y 85.422,Z 529.601,A -85,B 0,C 180,E1 -28128.863,E2 -28128.863} C_VEL
LIN {X 0,Y 78.32,Z 527.798,A -85,B 0,C 180,E1 -28137.448,E2 -28137.448} C_VEL
LIN {X 0,Y 73.669,Z 524.834,A -85,B 0,C 180,E1 -28147.59,E2 -28147.59} C_VEL
LIN {X 0,Y 71.827,Z 520.537,A -85,B 0,C 180,E1 -28158.736,E2 -28158.736} C_VEL
LIN {X 0,Y 71.912,Z 517.842,A -85,B 0,C 180,E1 -28164.412,E2 -28164.412} C_VEL
LIN {X 0,Y 71.868,Z 514.474,A -85,B 0,C 180,E1 -28170.021,E2 -28170.021} C_VEL
LIN {X 0,Y 71.841,Z 507.996,A -85,B 0,C 180,E1 -28178.459,E2 -28178.459} C_VEL
LIN {X 0,Y 72.883,Z 499.823,A -85,B 0,C 180,E1 -28186.836,E2 -28186.836} C_VEL
LIN {X 0,Y 74.755,Z 491.515,A -85,B 0,C 180,E1 -28193.571,E2 -28193.571} C_VEL
LIN {X 0,Y 76.431,Z 485.8,A -85,B 0,C 180,E1 -28197.392,E2 -28197.392} C_VEL
LIN {X 0,Y 76.536,Z 475.016,A -85,B 0,C 180,E1 -28203.455,E2 -28203.455} C_VEL
LIN {X 0,Y 76.709,Z 462.795,A -85,B 0,C 180,E1 -28209.111,E2 -28209.111} C_VEL
LIN {X 0,Y 76.918,Z 450.399,A -85,B 0,C 180,E1 -28213.686,E2 -28213.686} C_VEL
LIN {X 0,Y 76.845,Z 443.8,A -85,B 0,C 180,E1 -28215.778,E2 -28215.778} C_VEL
LIN {X 0,Y 75.142,Z 437.055,A -85,B 0,C 180,E1 -28218.205,E2 -28218.205} C_VEL
LIN {X 0,Y 72.834,Z 431.926,A -85,B 0,C 180,E1 -28220.327,E2 -28220.327} C_VEL
LIN {X 0,Y 72.709,Z 431.428,A -85,B 0,C 180,E1 -28220.678,E2 -28220.678} C_VEL
LIN {X 0,Y 72.416,Z 431.462,A -85,B 0,C 180,E1 -28230.966,E2 -28230.966} C_VEL
LIN {X 0,Y 72.391,Z 431.468,A -85,B 0,C 180,E1 -28237.144,E2 -28237.144} C_VEL
LIN {X 0,Y 72.702,Z 431.429,A -85,B 0,C 180,E1 -28245.242,E2 -28245.242} C_VEL
LIN {X 0,Y 72.844,Z 431.404,A -85,B 0,C 180,E1 -28248.869,E2 -28248.869} C_VEL
LIN {X 0,Y 73.565,Z 431.317,A -85,B 0,C 180,E1 -28259.995,E2 -28259.995} C_VEL
LIN {X 0,Y 72.831,Z 431.413,A -85,B 0,C 180,E1 -28271.123,E2 -28271.123} C_VEL
LIN {X 0,Y 72.527,Z 431.446,A -85,B 0,C 180,E1 -28276.895,E2 -28276.895} C_VEL
LIN {X 0,Y 72.39,Z 431.46,A -85,B 0,C 180,E1 -28282.846,E2 -28282.846} C_VEL
LIN {X 0,Y 72.375,Z 431.468,A -85,B 0,C 180,E1 -28289.041,E2 -28289.041} C_VEL
LIN {X 0,Y 72.306,Z 431.478,A -85,B 0,C 180,E1 -28295.669,E2 -28295.669} C_VEL
LIN {X 0,Y 72.257,Z 431.483,A -85,B 0,C 180,E1 -28302.903,E2 -28302.903} C_VEL
LIN {X 0,Y 72.301,Z 431.477,A -85,B 0,C 180,E1 -28311.036,E2 -28311.036} C_VEL
LIN {X 0,Y 72.3,Z 431.477,A -85,B 0,C 180,E1 -28314.298,E2 -28314.298} C_VEL
LIN {X 0,Y 72.364,Z 431.471,A -85,B 0,C 180,E1 -28320.926,E2 -28320.926} C_VEL
LIN {X 0,Y 72.397,Z 431.463,A -85,B 0,C 180,E1 -28327.13,E2 -28327.13} C_VEL
LIN {X 0,Y 72.722,Z 431.421,A -85,B 0,C 180,E1 -28335.089,E2 -28335.089} C_VEL
LIN {X 0,Y 72.857,Z 431.409,A -85,B 0,C 180,E1 -28338.856,E2 -28338.856} C_VEL
LIN {X 0,Y 73.565,Z 431.313,A -85,B 0,C 180,E1 -28349.98,E2 -28349.98} C_VEL
LIN {X 0,Y 72.865,Z 431.407,A -85,B 0,C 180,E1 -28361.101,E2 -28361.101} C_VEL
LIN {X 0,Y 72.775,Z 431.42,A -85,B 0,C 180,E1 -28363.785,E2 -28363.785} C_VEL
LIN {X 0,Y 76.398,Z 442.859,A -85,B 0,C 180,E1 -28368.618,E2 -28368.618} C_VEL
LIN {X 0,Y 78.863,Z 453.42,A -85,B 0,C 180,E1 -28373.273,E2 -28373.273} C_VEL
LIN {X 0,Y 79.156,Z 455.143,A -85,B 0,C 180,E1 -28374.067,E2 -28374.067} C_VEL
LIN {X 0,Y 79.246,Z 458.558,A -85,B 0,C 180,E1 -28375.539,E2 -28375.539} C_VEL
LIN {X 0,Y 78.468,Z 461.869,A -85,B 0,C 180,E1 -28376.914,E2 -28376.914} C_VEL
LIN {X 0,Y 77.074,Z 465.16,A -85,B 0,C 180,E1 -28378.252,E2 -28378.252} C_VEL
LIN {X 0,Y 75.295,Z 468.289,A -85,B 0,C 180,E1 -28379.59,E2 -28379.59} C_VEL
LIN {X 0,Y 69.449,Z 477.445,A -85,B 0,C 180,E1 -28384.457,E2 -28384.457} C_VEL
LIN {X 0,Y 68.148,Z 480.439,A -85,B 0,C 180,E1 -28386.515,E2 -28386.515} C_VEL
LIN {X 0,Y 65.653,Z 489.316,A -85,B 0,C 180,E1 -28393.741,E2 -28393.741} C_VEL
LIN {X 0,Y 63.843,Z 498.316,A -85,B 0,C 180,E1 -28403.137,E2 -28403.137} C_VEL
LIN {X 0,Y 63.142,Z 506.083,A -85,B 0,C 180,E1 -28413.569,E2 -28413.569} C_VEL
LIN {X 0,Y 64.217,Z 512.412,A -85,B 0,C 180,E1 -28424.13,E2 -28424.13} C_VEL
LIN {X 0,Y 67.293,Z 517.533,A -85,B 0,C 180,E1 -28434.011,E2 -28434.011} C_VEL
LIN {X 0,Y 72.099,Z 521.567,A -85,B 0,C 180,E1 -28442.799,E2 -28442.799} C_VEL
LIN {X 0,Y 78.61,Z 524.694,A -85,B 0,C 180,E1 -28450.558,E2 -28450.558} C_VEL
LIN {X 0,Y 88.985,Z 527.376,A -85,B 0,C 180,E1 -28458.66,E2 -28458.66} C_VEL
LIN {X 0,Y 100.528,Z 528.438,A -85,B 0,C 180,E1 -28464.693,E2 -28464.693} C_VEL
LIN {X 0,Y 110.887,Z 528.225,A -85,B 0,C 180,E1 -28468.62,E2 -28468.62} C_VEL
LIN {X 0,Y 109.729,Z 528.493,A -85,B 0,C 180,E1 -28469.707,E2 -28469.707} C_VEL
LIN {X 0,Y 100.555,Z 529.401,A -85,B 0,C 180,E1 -28473.027,E2 -28473.027} C_VEL
LIN {X 0,Y 89.713,Z 529.582,A -85,B 0,C 180,E1 -28478.457,E2 -28478.457} C_VEL
LIN {X 0,Y 80.246,Z 528.649,A -85,B 0,C 180,E1 -28485.548,E2 -28485.548} C_VEL
LIN {X 0,Y 72.514,Z 526.591,A -85,B 0,C 180,E1 -28494.469,E2 -28494.469} C_VEL
LIN {X 0,Y 67.296,Z 523.312,A -85,B 0,C 180,E1 -28505.333,E2 -28505.333} C_VEL
LIN {X 0,Y 65.093,Z 518.741,A -85,B 0,C 180,E1 -28517.553,E2 -28517.553} C_VEL
LIN {X 0,Y 65.126,Z 515.854,A -85,B 0,C 180,E1 -28523.828,E2 -28523.828} C_VEL
LIN {X 0,Y 65.001,Z 512.275,A -85,B 0,C 180,E1 -28530.023,E2 -28530.023} C_VEL
LIN {X 0,Y 64.971,Z 505.603,A -85,B 0,C 180,E1 -28539.171,E2 -28539.171} C_VEL
LIN {X 0,Y 66.328,Z 496.916,A -85,B 0,C 180,E1 -28548.557,E2 -28548.557} C_VEL
LIN {X 0,Y 68.45,Z 488.096,A -85,B 0,C 180,E1 -28555.895,E2 -28555.895} C_VEL
LIN {X 0,Y 69.365,Z 485.166,A -85,B 0,C 180,E1 -28557.967,E2 -28557.967} C_VEL
LIN {X 0,Y 69.536,Z 473.841,A -85,B 0,C 180,E1 -28564.935,E2 -28564.935} C_VEL
LIN {X 0,Y 69.864,Z 462.091,A -85,B 0,C 180,E1 -28570.86,E2 -28570.86} C_VEL
LIN {X 0,Y 70.241,Z 449.234,A -85,B 0,C 180,E1 -28576.011,E2 -28576.011} C_VEL
LIN {X 0,Y 70.046,Z 444.285,A -85,B 0,C 180,E1 -28577.783,E2 -28577.783} C_VEL
LIN {X 0,Y 68.32,Z 438.771,A -85,B 0,C 180,E1 -28580.138,E2 -28580.138} C_VEL
LIN {X 0,Y 65.609,Z 433.015,A -85,B 0,C 180,E1 -28582.941,E2 -28582.941} C_VEL
LIN {X 0,Y 65.47,Z 432.325,A -85,B 0,C 180,E1 -28583.33,E2 -28583.33} C_VEL
LIN {X 0,Y 65.3,Z 432.351,A -85,B 0,C 180,E1 -28589.471,E2 -28589.471} C_VEL
LIN {X 0,Y 65.255,Z 432.35,A -85,B 0,C 180,E1 -28594.475,E2 -28594.475} C_VEL
LIN {X 0,Y 65.595,Z 432.313,A -85,B 0,C 180,E1 -28604.719,E2 -28604.719} C_VEL
LIN {X 0,Y 65.74,Z 432.294,A -85,B 0,C 180,E1 -28607.649,E2 -28607.649} C_VEL
LIN {X 0,Y 66.462,Z 432.201,A -85,B 0,C 180,E1 -28619.995,E2 -28619.995} C_VEL
LIN {X 0,Y 65.732,Z 432.296,A -85,B 0,C 180,E1 -28632.342,E2 -28632.342} C_VEL
LIN {X 0,Y 65.358,Z 432.344,A -85,B 0,C 180,E1 -28638.814,E2 -28638.814} C_VEL
LIN {X 0,Y 65.236,Z 432.355,A -85,B 0,C 180,E1 -28645.52,E2 -28645.52} C_VEL
LIN {X 0,Y 65.185,Z 432.357,A -85,B 0,C 180,E1 -28652.614,E2 -28652.614} C_VEL
LIN {X 0,Y 65.193,Z 432.356,A -85,B 0,C 180,E1 -28660.975,E2 -28660.975} C_VEL
LIN {X 0,Y 65.209,Z 432.355,A -85,B 0,C 180,E1 -28669.682,E2 -28669.682} C_VEL
LIN {X 0,Y 65.231,Z 432.358,A -85,B 0,C 180,E1 -28679.522,E2 -28679.522} C_VEL
LIN {X 0,Y 65.234,Z 432.351,A -85,B 0,C 180,E1 -28684.449,E2 -28684.449} C_VEL
LIN {X 0,Y 65.619,Z 432.304,A -85,B 0,C 180,E1 -28694.543,E2 -28694.543} C_VEL
LIN {X 0,Y 65.754,Z 432.294,A -85,B 0,C 180,E1 -28697.634,E2 -28697.634} C_VEL
LIN {X 0,Y 66.488,Z 432.195,A -85,B 0,C 180,E1 -28709.978,E2 -28709.978} C_VEL
LIN {X 0,Y 65.814,Z 432.285,A -85,B 0,C 180,E1 -28721.137,E2 -28721.137} C_VEL
LIN {X 0,Y 69.9,Z 445.302,A -85,B 0,C 180,E1 -28727.533,E2 -28727.533} C_VEL
LIN {X 0,Y 72.242,Z 456.166,A -85,B 0,C 180,E1 -28732.878,E2 -28732.878} C_VEL
LIN {X 0,Y 73.251,Z 462.81,A -85,B 0,C 180,E1 -28736.319,E2 -28736.319} C_VEL
LIN {X 0,Y 72.893,Z 465.366,A -85,B 0,C 180,E1 -28737.599,E2 -28737.599} C_VEL
LIN {X 0,Y 69.504,Z 475.957,A -85,B 0,C 180,E1 -28743.476,E2 -28743.476} C_VEL
LIN {X 0,Y 68.148,Z 480.439,A -85,B 0,C 180,E1 -28746.515,E2 -28746.515} C_VEL
LIN {X 0,Y 66.201,Z 484.641,A -85,B 0,C 180,E1 -28749.65,E2 -28749.65} C_VEL
LIN {X 0,Y 61.638,Z 490.836,A -85,B 0,C 180,E1 -28755.273,E2 -28755.273} C_VEL
LIN {X 0,Y 57.543,Z 496.525,A -85,B 0,C 180,E1 -28762.136,E2 -28762.136} C_VEL
LIN {X 0,Y 56.42,Z 499.948,A -85,B 0,C 180,E1 -28766.921,E2 -28766.921} C_VEL
LIN {X 0,Y 56.355,Z 507.009,A -85,B 0,C 180,E1 -28778.037,E2 -28778.037} C_VEL
LIN {X 0,Y 58.525,Z 513.506,A -85,B 0,C 180,E1 -28790.116,E2 -28790.116} C_VEL
LIN {X 0,Y 63.243,Z 518.888,A -85,B 0,C 180,E1 -28801.404,E2 -28801.404} C_VEL
LIN {X 0,Y 70.673,Z 523.305,A -85,B 0,C 180,E1 -28811.477,E2 -28811.477} C_VEL
LIN {X 0,Y 81.203,Z 526.723,A -85,B 0,C 180,E1 -28820.259,E2 -28820.259} C_VEL
LIN {X 0,Y 87.162,Z 527.877,A -85,B 0,C 180,E1 -28823.78,E2 -28823.78} C_VEL
LIN {X 0,Y 97.741,Z 528.922,A -85,B 0,C 180,E1 -28828.568,E2 -28828.568} C_VEL
LIN {X 0,Y 96.872,Z 529.011,A -85,B 0,C 180,E1 -28829.506,E2 -28829.506} C_VEL
LIN {X 0,Y 85.5,Z 528.842,A -85,B 0,C 180,E1 -28834.748,E2 -28834.748} C_VEL
LIN {X 0,Y 75.382,Z 527.599,A -85,B 0,C 180,E1 -28841.799,E2 -28841.799} C_VEL
LIN {X 0,Y 66.965,Z 525.209,A -85,B 0,C 180,E1 -28851.002,E2 -28851.002} C_VEL
LIN {X 0,Y 61.072,Z 521.657,A -85,B 0,C 180,E1 -28862.621,E2 -28862.621} C_VEL
LIN {X 0,Y 58.442,Z 516.805,A -85,B 0,C 180,E1 -28876.11,E2 -28876.11} C_VEL
LIN {X 0,Y 58.372,Z 513.817,A -85,B 0,C 180,E1 -28883.11,E2 -28883.11} C_VEL
LIN {X 0,Y 58.131,Z 509.966,A -85,B 0,C 180,E1 -28890.025,E2 -28890.025} C_VEL
LIN {X 0,Y 58.147,Z 502.696,A -85,B 0,C 180,E1 -28900.466,E2 -28900.466} C_VEL
LIN {X 0,Y 59.779,Z 493.681,A -85,B 0,C 180,E1 -28910.678,E2 -28910.678} C_VEL
LIN {X 0,Y 62.29,Z 484.355,A -85,B 0,C 180,E1 -28918.68,E2 -28918.68} C_VEL
LIN {X 0,Y 62.535,Z 472.952,A -85,B 0,C 180,E1 -28926.428,E2 -28926.428} C_VEL
LIN {X 0,Y 63.046,Z 460.979,A -85,B 0,C 180,E1 -28933.011,E2 -28933.011} C_VEL
LIN {X 0,Y 63.621,Z 447.182,A -85,B 0,C 180,E1 -28939.005,E2 -28939.005} C_VEL
LIN {X 0,Y 62.192,Z 441.994,A -85,B 0,C 180,E1 -28941.565,E2 -28941.565} C_VEL
LIN {X 0,Y 58.347,Z 433.687,A -85,B 0,C 180,E1 -28946.448,E2 -28946.448} C_VEL
LIN {X 0,Y 58.275,Z 433.221,A -85,B 0,C 180,E1 -28946.769,E2 -28946.769} C_VEL
LIN {X 0,Y 58.185,Z 433.234,A -85,B 0,C 180,E1 -28951.102,E2 -28951.102} C_VEL
LIN {X 0,Y 58.187,Z 433.236,A -85,B 0,C 180,E1 -28958.749,E2 -28958.749} C_VEL
LIN {X 0,Y 58.609,Z 433.185,A -85,B 0,C 180,E1 -28966.117,E2 -28966.117} C_VEL
LIN {X 0,Y 58.799,Z 433.16,A -85,B 0,C 180,E1 -28973.129,E2 -28973.129} C_VEL
LIN {X 0,Y 59.354,Z 433.086,A -85,B 0,C 180,E1 -28979.994,E2 -28979.994} C_VEL
LIN {X 0,Y 58.78,Z 433.154,A -85,B 0,C 180,E1 -28986.861,E2 -28986.861} C_VEL
LIN {X 0,Y 58.477,Z 433.193,A -85,B 0,C 180,E1 -28995.871,E2 -28995.871} C_VEL
LIN {X 0,Y 58.178,Z 433.234,A -85,B 0,C 180,E1 -29001.241,E2 -29001.241} C_VEL
LIN {X 0,Y 58.144,Z 433.241,A -85,B 0,C 180,E1 -29008.906,E2 -29008.906} C_VEL
LIN {X 0,Y 58.036,Z 433.255,A -85,B 0,C 180,E1 -29017.256,E2 -29017.256} C_VEL
LIN {X 0,Y 58.02,Z 433.253,A -85,B 0,C 180,E1 -29026.608,E2 -29026.608} C_VEL
LIN {X 0,Y 58.03,Z 433.257,A -85,B 0,C 180,E1 -29032.701,E2 -29032.701} C_VEL
LIN {X 0,Y 58.136,Z 433.244,A -85,B 0,C 180,E1 -29041.054,E2 -29041.054} C_VEL
LIN {X 0,Y 58.512,Z 433.188,A -85,B 0,C 180,E1 -29053.901,E2 -29053.901} C_VEL
LIN {X 0,Y 58.797,Z 433.154,A -85,B 0,C 180,E1 -29063.11,E2 -29063.11} C_VEL
LIN {X 0,Y 59.378,Z 433.08,A -85,B 0,C 180,E1 -29069.975,E2 -29069.975} C_VEL
LIN {X 0,Y 58.796,Z 433.153,A -85,B 0,C 180,E1 -29077.919,E2 -29077.919} C_VEL
LIN {X 0,Y 62.209,Z 443.472,A -85,B 0,C 180,E1 -29083.866,E2 -29083.866} C_VEL
LIN {X 0,Y 64.204,Z 451.425,A -85,B 0,C 180,E1 -29088.318,E2 -29088.318} C_VEL
LIN {X 0,Y 65.889,Z 460.615,A -85,B 0,C 180,E1 -29093.552,E2 -29093.552} C_VEL
LIN {X 0,Y 66.274,Z 464.089,A -85,B 0,C 180,E1 -29095.575,E2 -29095.575} C_VEL
LIN {X 0,Y 62.994,Z 474.111,A -85,B 0,C 180,E1 -29101.398,E2 -29101.398} C_VEL
LIN {X 0,Y 59.571,Z 485.052,A -85,B 0,C 180,E1 -29109.938,E2 -29109.938} C_VEL
LIN {X 0,Y 57.347,Z 494.152,A -85,B 0,C 180,E1 -29119.345,E2 -29119.345} C_VEL
LIN {X 0,Y 56.42,Z 499.948,A -85,B 0,C 180,E1 -29126.921,E2 -29126.921} C_VEL
LIN {X 0,Y 55.563,Z 503.177,A -85,B 0,C 180,E1 -29131.904,E2 -29131.904} C_VEL
LIN {X 0,Y 53.195,Z 507.712,A -85,B 0,C 180,E1 -29140.867,E2 -29140.867} C_VEL
LIN {X 0,Y 52.161,Z 511.723,A -85,B 0,C 180,E1 -29150.771,E2 -29150.771} C_VEL
LIN {X 0,Y 53.322,Z 514.128,A -85,B 0,C 180,E1 -29156.556,E2 -29156.556} C_VEL
LIN {X 0,Y 58.489,Z 518.873,A -85,B 0,C 180,E1 -29166.907,E2 -29166.907} C_VEL
LIN {X 0,Y 65.688,Z 522.854,A -85,B 0,C 180,E1 -29175.743,E2 -29175.743} C_VEL
LIN {X 0,Y 77.245,Z 526.682,A -85,B 0,C 180,E1 -29184.568,E2 -29184.568} C_VEL
LIN {X 0,Y 84.428,Z 528.11,A -85,B 0,C 180,E1 -29188.316,E2 -29188.316} C_VEL
LIN {X 0,Y 81.686,Z 528.024,A -85,B 0,C 180,E1 -29190.681,E2 -29190.681} C_VEL
LIN {X 0,Y 70.896,Z 526.46,A -85,B 0,C 180,E1 -29197.565,E2 -29197.565} C_VEL
LIN {X 0,Y 61.696,Z 523.762,A -85,B 0,C 180,E1 -29206.918,E2 -29206.918} C_VEL
LIN {X 0,Y 55.04,Z 519.895,A -85,B 0,C 180,E1 -29219.318,E2 -29219.318} C_VEL
LIN {X 0,Y 51.894,Z 514.723,A -85,B 0,C 180,E1 -29234.315,E2 -29234.315} C_VEL
LIN {X 0,Y 51.672,Z 511.537,A -85,B 0,C 180,E1 -29242.212,E2 -29242.212} C_VEL
LIN {X 0,Y 51.287,Z 507.516,A -85,B 0,C 180,E1 -29250.029,E2 -29250.029} C_VEL
LIN {X 0,Y 51.226,Z 501.259,A -85,B 0,C 180,E1 -29259.904,E2 -29259.904} C_VEL
LIN {X 0,Y 52.7,Z 492.922,A -85,B 0,C 180,E1 -29270.457,E2 -29270.457} C_VEL
LIN {X 0,Y 55.233,Z 483.439,A -85,B 0,C 180,E1 -29279.572,E2 -29279.572} C_VEL
LIN {X 0,Y 55.567,Z 472.248,A -85,B 0,C 180,E1 -29288.099,E2 -29288.099} C_VEL
LIN {X 0,Y 56.266,Z 460.861,A -85,B 0,C 180,E1 -29295.119,E2 -29295.119} C_VEL
LIN {X 0,Y 56.995,Z 448.296,A -85,B 0,C 180,E1 -29301.309,E2 -29301.309} C_VEL
LIN {X 0,Y 55.592,Z 444.048,A -85,B 0,C 180,E1 -29303.953,E2 -29303.953} C_VEL
LIN {X 0,Y 51.389,Z 435.248,A -85,B 0,C 180,E1 -29310.272,E2 -29310.272} C_VEL
LIN {X 0,Y 51.13,Z 434.111,A -85,B 0,C 180,E1 -29311.236,E2 -29311.236} C_VEL
LIN {X 0,Y 51.391,Z 434.08,A -85,B 0,C 180,E1 -29324.12,E2 -29324.12} C_VEL
LIN {X 0,Y 51.673,Z 434.043,A -85,B 0,C 180,E1 -29332.176,E2 -29332.176} C_VEL
LIN {X 0,Y 52.239,Z 433.971,A -85,B 0,C 180,E1 -29339.993,E2 -29339.993} C_VEL
LIN {X 0,Y 51.659,Z 434.042,A -85,B 0,C 180,E1 -29347.812,E2 -29347.812} C_VEL
LIN {X 0,Y 51.357,Z 434.081,A -85,B 0,C 180,E1 -29356.587,E2 -29356.587} C_VEL
LIN {X 0,Y 51.018,Z 434.121,A -85,B 0,C 180,E1 -29364.402,E2 -29364.402} C_VEL
LIN {X 0,Y 51.026,Z 434.125,A -85,B 0,C 180,E1 -29374.22,E2 -29374.22} C_VEL
LIN {X 0,Y 50.987,Z 434.129,A -85,B 0,C 180,E1 -29386.396,E2 -29386.396} C_VEL
LIN {X 0,Y 51.02,Z 434.121,A -85,B 0,C 180,E1 -29396.531,E2 -29396.531} C_VEL
LIN {X 0,Y 51.017,Z 434.121,A -85,B 0,C 180,E1 -29405.558,E2 -29405.558} C_VEL
LIN {X 0,Y 51.459,Z 434.066,A -85,B 0,C 180,E1 -29414.119,E2 -29414.119} C_VEL
LIN {X 0,Y 51.673,Z 434.039,A -85,B 0,C 180,E1 -29422.154,E2 -29422.154} C_VEL
LIN {X 0,Y 52.261,Z 433.966,A -85,B 0,C 180,E1 -29429.972,E2 -29429.972} C_VEL
LIN {X 0,Y 51.916,Z 434.018,A -85,B 0,C 180,E1 -29433.852,E2 -29433.852} C_VEL
LIN {X 0,Y 54.925,Z 442.898,A -85,B 0,C 180,E1 -29440.106,E2 -29440.106} C_VEL
LIN {X 0,Y 57.316,Z 452.039,A -85,B 0,C 180,E1 -29445.988,E2 -29445.988} C_VEL
LIN {X 0,Y 58.894,Z 461.109,A -85,B 0,C 180,E1 -29451.868,E2 -29451.868} C_VEL
LIN {X 0,Y 59.238,Z 463.668,A -85,B 0,C 180,E1 -29453.576,E2 -29453.576} C_VEL
LIN {X 0,Y 58.433,Z 467.015,A -85,B 0,C 180,E1 -29455.585,E2 -29455.585} C_VEL
LIN {X 0,Y 54.628,Z 477.953,A -85,B 0,C 180,E1 -29463.268,E2 -29463.268} C_VEL
LIN {X 0,Y 51.33,Z 488.706,A -85,B 0,C 180,E1 -29473.905,E2 -29473.905} C_VEL
LIN {X 0,Y 49.607,Z 497.472,A -85,B 0,C 180,E1 -29485.489,E2 -29485.489} C_VEL
LIN {X 0,Y 49.36,Z 504.378,A -85,B 0,C 180,E1 -29496.957,E2 -29496.957} C_VEL
LIN {X 0,Y 51.127,Z 510.795,A -85,B 0,C 180,E1 -29509.516,E2 -29509.516} C_VEL
LIN {X 0,Y 53.322,Z 514.128,A -85,B 0,C 180,E1 -29516.556,E2 -29516.556} C_VEL
LIN {X 0,Y 54.992,Z 516.416,A -85,B 0,C 180,E1 -29522.059,E2 -29522.059} C_VEL
LIN {X 0,Y 57.338,Z 519.513,A -85,B 0,C 180,E1 -29531.38,E2 -29531.38} C_VEL
LIN {X 0,Y 60.213,Z 521.68,A -85,B 0,C 180,E1 -29538.304,E2 -29538.304} C_VEL
LIN {X 0,Y 63.557,Z 523.27,A -85,B 0,C 180,E1 -29542.584,E2 -29542.584} C_VEL
LIN {X 0,Y 64.942,Z 523.799,A -85,B 0,C 180,E1 -29543.743,E2 -29543.743} C_VEL
LIN {X 0,Y 72.889,Z 526.295,A -85,B 0,C 180,E1 -29548.828,E2 -29548.828} C_VEL
LIN {X 0,Y 61.599,Z 523.796,A -85,B 0,C 180,E1 -29557.041,E2 -29557.041} C_VEL
LIN {X 0,Y 52.67,Z 520.249,A -85,B 0,C 180,E1 -29568.19,E2 -29568.19} C_VEL
LIN {X 0,Y 46.797,Z 515.459,A -85,B 0,C 180,E1 -29583.258,E2 -29583.258} C_VEL
LIN {X 0,Y 45.106,Z 510.934,A -85,B 0,C 180,E1 -29596.518,E2 -29596.518} C_VEL
LIN {X 0,Y 44.879,Z 508.175,A -85,B 0,C 180,E1 -29603.288,E2 -29603.288} C_VEL
LIN {X 0,Y 44.335,Z 503.61,A -85,B 0,C 180,E1 -29612.304,E2 -29612.304} C_VEL
LIN {X 0,Y 44.95,Z 495.158,A -85,B 0,C 180,E1 -29625.913,E2 -29625.913} C_VEL
LIN {X 0,Y 47.059,Z 486.517,A -85,B 0,C 180,E1 -29636.652,E2 -29636.652} C_VEL
LIN {X 0,Y 48.157,Z 482.462,A -85,B 0,C 180,E1 -29640.751,E2 -29640.751} C_VEL
LIN {X 0,Y 48.576,Z 472.642,A -85,B 0,C 180,E1 -29649.308,E2 -29649.308} C_VEL
LIN {X 0,Y 49.579,Z 460.603,A -85,B 0,C 180,E1 -29657.783,E2 -29657.783} C_VEL
LIN {X 0,Y 50.367,Z 449.711,A -85,B 0,C 180,E1 -29663.949,E2 -29663.949} C_VEL
LIN {X 0,Y 47.276,Z 442.424,A -85,B 0,C 180,E1 -29669.878,E2 -29669.878} C_VEL
LIN {X 0,Y 45.924,Z 439.3,A -85,B 0,C 180,E1 -29672.662,E2 -29672.662} C_VEL
LIN {X 0,Y 44.42,Z 436.64,A -85,B 0,C 180,E1 -29675.452,E2 -29675.452} C_VEL
LIN {X 0,Y 43.978,Z 435.007,A -85,B 0,C 180,E1 -29677.066,E2 -29677.066} C_VEL
LIN {X 0,Y 44.195,Z 434.971,A -85,B 0,C 180,E1 -29682.687,E2 -29682.687} C_VEL
LIN {X 0,Y 44.512,Z 434.931,A -85,B 0,C 180,E1 -29690.908,E2 -29690.908} C_VEL
LIN {X 0,Y 45.114,Z 434.858,A -85,B 0,C 180,E1 -29699.992,E2 -29699.992} C_VEL
LIN {X 0,Y 44.508,Z 434.936,A -85,B 0,C 180,E1 -29709.077,E2 -29709.077} C_VEL
LIN {X 0,Y 44.126,Z 434.988,A -85,B 0,C 180,E1 -29718.566,E2 -29718.566} C_VEL
LIN {X 0,Y 43.831,Z 435.024,A -85,B 0,C 180,E1 -29728.743,E2 -29728.743} C_VEL
LIN {X 0,Y 43.844,Z 435.023,A -85,B 0,C 180,E1 -29736.674,E2 -29736.674} C_VEL
LIN {X 0,Y 43.795,Z 435.022,A -85,B 0,C 180,E1 -29750.024,E2 -29750.024} C_VEL
LIN {X 0,Y 43.825,Z 435.026,A -85,B 0,C 180,E1 -29761.206,E2 -29761.206} C_VEL
LIN {X 0,Y 44.23,Z 434.967,A -85,B 0,C 180,E1 -29772.409,E2 -29772.409} C_VEL
LIN {X 0,Y 44.527,Z 434.93,A -85,B 0,C 180,E1 -29780.885,E2 -29780.885} C_VEL
LIN {X 0,Y 45.018,Z 434.932,A -85,B 0,C 180,E1 -29788.569,E2 -29788.569} C_VEL
LIN {X 0,Y 48.508,Z 444.85,A -85,B 0,C 180,E1 -29797.252,E2 -29797.252} C_VEL
LIN {X 0,Y 50.636,Z 453.726,A -85,B 0,C 180,E1 -29804.027,E2 -29804.027} C_VEL
LIN {X 0,Y 52.077,Z 462.682,A -85,B 0,C 180,E1 -29810.717,E2 -29810.717} C_VEL
LIN {X 0,Y 52.212,Z 464.996,A -85,B 0,C 180,E1 -29812.41,E2 -29812.41} C_VEL
LIN {X 0,Y 48.014,Z 476.275,A -85,B 0,C 180,E1 -29820.909,E2 -29820.909} C_VEL
LIN {X 0,Y 44.677,Z 486.405,A -85,B 0,C 180,E1 -29831.664,E2 -29831.664} C_VEL
LIN {X 0,Y 42.694,Z 495.862,A -85,B 0,C 180,E1 -29845.329,E2 -29845.329} C_VEL
LIN {X 0,Y 42.511,Z 502.77,A -85,B 0,C 180,E1 -29858.172,E2 -29858.172} C_VEL
LIN {X 0,Y 44.819,Z 509.772,A -85,B 0,C 180,E1 -29873.254,E2 -29873.254} C_VEL
LIN {X 0,Y 50.799,Z 516.369,A -85,B 0,C 180,E1 -29887.959,E2 -29887.959} C_VEL
LIN {X 0,Y 60.75,Z 522.146,A -85,B 0,C 180,E1 -29900.314,E2 -29900.314} C_VEL
LIN {X 0,Y 64.942,Z 523.799,A -85,B 0,C 180,E1 -29903.743,E2 -29903.743} C_VEL
LIN {X 0,Y 65.383,Z 524.083,A -85,B 0,C 180,E1 -29904.819,E2 -29904.819} C_VEL
LIN {X 0,Y 64.62,Z 524.089,A -85,B 0,C 180,E1 -29906.901,E2 -29906.901} C_VEL
LIN {X 0,Y 62.28,Z 523.62,A -85,B 0,C 180,E1 -29909.445,E2 -29909.445} C_VEL
LIN {X 0,Y 55.687,Z 521.638,A -85,B 0,C 180,E1 -29914.042,E2 -29914.042} C_VEL
LIN {X 0,Y 50.498,Z 519.651,A -85,B 0,C 180,E1 -29918.888,E2 -29918.888} C_VEL
LIN {X 0,Y 42.227,Z 514.677,A -85,B 0,C 180,E1 -29934.417,E2 -29934.417} C_VEL
LIN {X 0,Y 38.662,Z 508.499,A -85,B 0,C 180,E1 -29954.217,E2 -29954.217} C_VEL
LIN {X 0,Y 38.245,Z 505.625,A -85,B 0,C 180,E1 -29962.117,E2 -29962.117} C_VEL
LIN {X 0,Y 37.451,Z 499.344,A -85,B 0,C 180,E1 -29975.423,E2 -29975.423} C_VEL
LIN {X 0,Y 38.817,Z 490.024,A -85,B 0,C 180,E1 -29991.27,E2 -29991.27} C_VEL
LIN {X 0,Y 41.044,Z 482.35,A -85,B 0,C 180,E1 -30001.096,E2 -30001.096} C_VEL
LIN {X 0,Y 41.607,Z 472.771,A -85,B 0,C 180,E1 -30010.929,E2 -30010.929} C_VEL
LIN {X 0,Y 42.959,Z 460.548,A -85,B 0,C 180,E1 -30020.95,E2 -30020.95} C_VEL
LIN {X 0,Y 43.844,Z 452.595,A -85,B 0,C 180,E1 -30026.19,E2 -30026.19} C_VEL
LIN {X 0,Y 42.99,Z 449.555,A -85,B 0,C 180,E1 -30028.921,E2 -30028.921} C_VEL
LIN {X 0,Y 39.932,Z 442.473,A -85,B 0,C 180,E1 -30036.662,E2 -30036.662} C_VEL
LIN {X 0,Y 37.213,Z 436.298,A -85,B 0,C 180,E1 -30044.45,E2 -30044.45} C_VEL
LIN {X 0,Y 37.172,Z 435.853,A -85,B 0,C 180,E1 -30045.216,E2 -30045.216} C_VEL
LIN {X 0,Y 37.974,Z 435.747,A -85,B 0,C 180,E1 -30059.991,E2 -30059.991} C_VEL
LIN {X 0,Y 37.307,Z 435.838,A -85,B 0,C 180,E1 -30070.848,E2 -30070.848} C_VEL
LIN {X 0,Y 37.049,Z 435.868,A -85,B 0,C 180,E1 -30078.353,E2 -30078.353} C_VEL
LIN {X 0,Y 36.722,Z 435.908,A -85,B 0,C 180,E1 -30095.028,E2 -30095.028} C_VEL
LIN {X 0,Y 36.729,Z 435.9,A -85,B 0,C 180,E1 -30099.998,E2 -30099.998} C_VEL
LIN {X 0,Y 36.72,Z 435.903,A -85,B 0,C 180,E1 -30109.943,E2 -30109.943} C_VEL
LIN {X 0,Y 36.705,Z 435.906,A -85,B 0,C 180,E1 -30114.893,E2 -30114.893} C_VEL
LIN {X 0,Y 37.056,Z 435.863,A -85,B 0,C 180,E1 -30131.464,E2 -30131.464} C_VEL
LIN {X 0,Y 37.372,Z 435.823,A -85,B 0,C 180,E1 -30139.806,E2 -30139.806} C_VEL
LIN {X 0,Y 37.91,Z 437.441,A -85,B 0,C 180,E1 -30141.969,E2 -30141.969} C_VEL
LIN {X 0,Y 40.282,Z 440.894,A -85,B 0,C 180,E1 -30147.463,E2 -30147.463} C_VEL
LIN {X 0,Y 42.638,Z 448.762,A -85,B 0,C 180,E1 -30155.419,E2 -30155.419} C_VEL
LIN {X 0,Y 44.254,Z 456.641,A -85,B 0,C 180,E1 -30162.578,E2 -30162.578} C_VEL
LIN {X 0,Y 45.266,Z 464.142,A -85,B 0,C 180,E1 -30169.223,E2 -30169.223} C_VEL
LIN {X 0,Y 45.017,Z 465.801,A -85,B 0,C 180,E1 -30170.517,E2 -30170.517} C_VEL
LIN {X 0,Y 40.081,Z 478.295,A -85,B 0,C 180,E1 -30181.694,E2 -30181.694} C_VEL
LIN {X 0,Y 36.987,Z 487.928,A -85,B 0,C 180,E1 -30194.491,E2 -30194.491} C_VEL
LIN {X 0,Y 35.551,Z 496.626,A -85,B 0,C 180,E1 -30210.394,E2 -30210.394} C_VEL
LIN {X 0,Y 36.745,Z 504.811,A -85,B 0,C 180,E1 -30228.983,E2 -30228.983} C_VEL
LIN {X 0,Y 41.122,Z 511.422,A -85,B 0,C 180,E1 -30244.752,E2 -30244.752} C_VEL
LIN {X 0,Y 48.033,Z 516.914,A -85,B 0,C 180,E1 -30257.023,E2 -30257.023} C_VEL
LIN {X 0,Y 59.618,Z 522.683,A -85,B 0,C 180,E1 -30268.14,E2 -30268.14} C_VEL
LIN {X 0,Y 57.683,Z 522.232,A -85,B 0,C 180,E1 -30271.526,E2 -30271.526} C_VEL
LIN {X 0,Y 50.498,Z 519.651,A -85,B 0,C 180,E1 -30278.888,E2 -30278.888} C_VEL
LIN {X 0,Y 46.507,Z 517.785,A -85,B 0,C 180,E1 -30283.512,E2 -30283.512} C_VEL
LIN {X 0,Y 39.695,Z 513.689,A -85,B 0,C 180,E1 -30291.349,E2 -30291.349} C_VEL
LIN {X 0,Y 34.093,Z 508.964,A -85,B 0,C 180,E1 -30301.84,E2 -30301.84} C_VEL
LIN {X 0,Y 32.386,Z 506.106,A -85,B 0,C 180,E1 -30310.409,E2 -30310.409} C_VEL
LIN {X 0,Y 31.622,Z 502.832,A -85,B 0,C 180,E1 -30320.452,E2 -30320.452} C_VEL
LIN {X 0,Y 30.666,Z 496.145,A -85,B 0,C 180,E1 -30336.628,E2 -30336.628} C_VEL
LIN {X 0,Y 32.002,Z 488.123,A -85,B 0,C 180,E1 -30352.651,E2 -30352.651} C_VEL
LIN {X 0,Y 33.838,Z 482.163,A -85,B 0,C 180,E1 -30361.695,E2 -30361.695} C_VEL
LIN {X 0,Y 34.685,Z 472.899,A -85,B 0,C 180,E1 -30373.203,E2 -30373.203} C_VEL
LIN {X 0,Y 36.543,Z 460.105,A -85,B 0,C 180,E1 -30385.59,E2 -30385.59} C_VEL
LIN {X 0,Y 37.406,Z 453.903,A -85,B 0,C 180,E1 -30390.438,E2 -30390.438} C_VEL
LIN {X 0,Y 34.228,Z 445.681,A -85,B 0,C 180,E1 -30401.331,E2 -30401.331} C_VEL
LIN {X 0,Y 32.686,Z 441.821,A -85,B 0,C 180,E1 -30407.573,E2 -30407.573} C_VEL
